fb_balkon_peryla_send(str_Rec:=fb_KL6301_0.str_Data_Rec, bData:=balkon_peryla,  Group_Address:=balkon_peryla_adr, bsend:=((fb_balkon_peryla_send.bData XOR fb_balkon_peryla_read.bData XOR balkon_peryla)OR fb_heartbeat2_timer.q));   (*       balkon_peryla_read.bData XOR balkon_peryla)) AND fb_heartbeat2_timer.q))      )));*)
IF NOT fb_balkon_peryla_read.bDataReceive OR  fb_heartbeat2_timer.q THEN fb_balkon_peryla_send.bSend:=FALSE; fb_balkon_peryla_send(str_Rec:=fb_KL6301_0.str_Data_Rec, bData:=balkon_peryla,  Group_Address:=balkon_peryla_adr);END_IF
fb_kino_l_send(str_Rec:=fb_KL6301_0.str_Data_Rec, bData:=kino_l,  Group_Address:=kino_l_adr, bsend:=((fb_kino_l_send.bData  <>  fb_kino_l_read.bData <> kino_l)OR fb_heartbeat2_timer.q));
IF NOT fb_kino_l_read.bDataReceive OR  fb_heartbeat2_timer.q THEN fb_kino_l_send.bSend:=FALSE; fb_kino_l_send(str_Rec:=fb_KL6301_0.str_Data_Rec,  Group_Address:=kino_l_adr);END_IF
fb_balkon_bra_send(str_Rec:=fb_KL6301_0.str_Data_Rec, bData:=balkon_bra,  Group_Address:=balkon_bra_adr, bsend:=((fb_balkon_bra_read.bData  XOR fb_balkon_bra_read.bData XOR balkon_bra)OR fb_heartbeat2_timer.q));   (*       balkon_bra_read.bData XOR balkon_bra)) AND fb_heartbeat2_timer.q))      )));*)
IF NOT fb_balkon_bra_read.bDataReceive OR  fb_heartbeat2_timer.q THEN fb_balkon_bra_send.bSend:=FALSE; fb_balkon_bra_send(str_Rec:=fb_KL6301_0.str_Data_Rec, bData:=balkon_bra,  Group_Address:=balkon_bra_adr);END_IF
fb_kabinet_balkon_l_send(str_Rec:=fb_KL6301_0.str_Data_Rec, bData:=kabinet_balkon_l,  Group_Address:=kabinet_balkon_l_adr, bsend:=(( fb_kabinet_balkon_l_send.bData XOR fb_kabinet_balkon_l_read.bData XOR kabinet_balkon_l)OR fb_heartbeat2_timer.q));   (*       kabinet_balkon_l_read.bData XOR kabinet_balkon_l)) AND fb_heartbeat2_timer.q))      )));*)
IF NOT fb_kabinet_balkon_l_read.bDataReceive OR  fb_heartbeat2_timer.q THEN fb_kabinet_balkon_l_send.bSend:=FALSE; fb_kabinet_balkon_l_send(str_Rec:=fb_KL6301_0.str_Data_Rec, bData:=kabinet_balkon_l,  Group_Address:=kabinet_balkon_l_adr);END_IF
fb_balkon_send(str_Rec:=fb_KL6301_0.str_Data_Rec, bData:=balkon,  Group_Address:=balkon_adr, bsend:=((fb_balkon_send.bData XOR fb_balkon_read.bData XOR balkon)OR fb_heartbeat2_timer.q));   (*       balkon_read.bData XOR balkon)) AND fb_heartbeat2_timer.q))      )));*)
IF NOT fb_balkon_read.bDataReceive OR  fb_heartbeat2_timer.q THEN fb_balkon_send.bSend:=FALSE; fb_balkon_send(str_Rec:=fb_KL6301_0.str_Data_Rec, bData:=balkon,  Group_Address:=balkon_adr);END_IF
fb_korydor1_send(str_Rec:=fb_KL6301_0.str_Data_Rec, bData:=korydor1,  Group_Address:=korydor1_adr, bsend:=((fb_korydor1_send.bData XOR fb_korydor1_read.bData XOR korydor1)OR fb_heartbeat2_timer.q));   (* *)
IF NOT fb_korydor1_read.bDataReceive OR  fb_heartbeat2_timer.q THEN fb_korydor1_send.bSend:=FALSE; fb_korydor1_send(str_Rec:=fb_KL6301_0.str_Data_Rec, bData:=korydor1,  Group_Address:=korydor1_adr);END_IF
fb_kino_bra_send(str_Rec:=fb_KL6301_0.str_Data_Rec, bData:=kino_bra,  Group_Address:=kino_bra_adr, bsend:=((fb_kino_bra_send.bData XOR fb_kino_bra_read.bData XOR kino_bra)OR fb_heartbeat2_timer.q));
IF NOT fb_kino_bra_read.bDataReceive OR  fb_heartbeat2_timer.q THEN fb_kino_bra_send.bSend:=FALSE; fb_kino_bra_send(str_Rec:=fb_KL6301_0.str_Data_Rec, bData:=kino_bra,  Group_Address:=kino_bra_adr);END_IF
fb_korydor2_send(str_Rec:=fb_KL6301_0.str_Data_Rec, bData:=korydor2,  Group_Address:=korydor2_adr, bsend:=((fb_korydor2_send.bData XOR fb_korydor2_read.bData XOR korydor2)OR fb_heartbeat2_timer.q));
IF NOT fb_korydor2_read.bDataReceive OR  fb_heartbeat2_timer.q THEN fb_korydor2_send.bSend:=FALSE; fb_korydor2_send(str_Rec:=fb_KL6301_0.str_Data_Rec, bData:=korydor2,  Group_Address:=korydor2_adr);END_IF
fb_studio_pidsvitka_send(str_Rec:=fb_KL6301_0.str_Data_Rec, bData:=studio_pidsvitka,  Group_Address:=studio_pidsvitka_adr, bsend:=((fb_studio_pidsvitka_send.bData XOR fb_studio_pidsvitka_read.bData XOR studio_pidsvitka)OR fb_heartbeat2_timer.q));
IF NOT fb_studio_pidsvitka_read.bDataReceive OR  fb_heartbeat2_timer.q THEN fb_studio_pidsvitka_send.bSend:=FALSE; fb_studio_pidsvitka_send(str_Rec:=fb_KL6301_0.str_Data_Rec, bData:=studio_pidsvitka,  Group_Address:=studio_pidsvitka_adr);END_IF
fb_skhody2_3_send(str_Rec:=fb_KL6301_0.str_Data_Rec, bData:=skhody2_3,  Group_Address:=skhody2_3_adr, bsend:=((fb_skhody2_3_send.bData XOR fb_skhody2_3_read.bData XOR skhody2_3)OR fb_heartbeat2_timer.q));
IF NOT fb_skhody2_3_read.bDataReceive OR  fb_heartbeat2_timer.q THEN fb_skhody2_3_send.bSend:=FALSE; fb_skhody2_3_send(str_Rec:=fb_KL6301_0.str_Data_Rec, bData:=skhody2_3,  Group_Address:=skhody2_3_adr);END_IF
fb_studio_l_send(str_Rec:=fb_KL6301_0.str_Data_Rec, bData:=studio_l,  Group_Address:=studio_l_adr, bsend:=((fb_studio_l_send.bData XOR fb_studio_l_read.bData XOR studio_l)OR fb_heartbeat2_timer.q));
IF NOT fb_studio_l_read.bDataReceive OR  fb_heartbeat2_timer.q THEN fb_studio_l_send.bSend:=FALSE; fb_studio_l_send(str_Rec:=fb_KL6301_0.str_Data_Rec, bData:=studio_l,  Group_Address:=studio_l_adr);END_IF
fb_kabinet_pidsvitka_kolo_send(str_Rec:=fb_KL6301_0.str_Data_Rec, bData:=kabinet_pidsvitka_kolo,  Group_Address:=kabinet_pidsvitka_kolo_adr, bsend:=((fb_kabinet_pidsvitka_kolo_send.bData XOR fb_kabinet_pidsvitka_kolo_read.bData XOR kabinet_pidsvitka_kolo)OR fb_heartbeat2_timer.q));
IF NOT fb_kabinet_pidsvitka_kolo_read.bDataReceive OR  fb_heartbeat2_timer.q THEN fb_kabinet_pidsvitka_kolo_send.bSend:=FALSE; fb_kabinet_pidsvitka_kolo_send(str_Rec:=fb_KL6301_0.str_Data_Rec, bData:=kabinet_pidsvitka_kolo,  Group_Address:=kabinet_pidsvitka_kolo_adr);END_IF
fb_kabinet_svitlo_send(str_Rec:=fb_KL6301_0.str_Data_Rec, bData:=kabinet_svitlo,  Group_Address:=kabinet_svitlo_adr, bsend:=((fb_kabinet_svitlo_send.bData XOR fb_kabinet_svitlo_read.bData XOR kabinet_svitlo)OR fb_heartbeat2_timer.q));
IF NOT fb_kabinet_svitlo_read.bDataReceive OR  fb_heartbeat2_timer.q THEN fb_kabinet_svitlo_send.bSend:=FALSE; fb_kabinet_svitlo_send(str_Rec:=fb_KL6301_0.str_Data_Rec, bData:=kabinet_svitlo,  Group_Address:=kabinet_svitlo_adr);END_IF
fb_stend_send(str_Rec:=fb_KL6301_0.str_Data_Rec, bData:=stend,  Group_Address:=stend_adr, bsend:=((fb_stend_send.bData XOR fb_stend_read.bData XOR stend)OR fb_heartbeat2_timer.q));
IF NOT fb_stend_read.bDataReceive OR  fb_heartbeat2_timer.q THEN fb_stend_send.bSend:=FALSE; fb_stend_send(str_Rec:=fb_KL6301_0.str_Data_Rec, bData:=stend,  Group_Address:=stend_adr);END_IF
fb_kabinet_kobra_send(str_Rec:=fb_KL6301_0.str_Data_Rec, bData:=kabinet_kobra,  Group_Address:=kabinet_kobra_adr, bsend:=((fb_kabinet_kobra_send.bData XOR fb_kabinet_kobra_read.bData XOR kabinet_kobra)OR fb_heartbeat2_timer.q));
IF NOT fb_kabinet_kobra_read.bDataReceive OR  fb_heartbeat2_timer.q THEN fb_kabinet_kobra_send.bSend:=FALSE; fb_kabinet_kobra_send(str_Rec:=fb_KL6301_0.str_Data_Rec, bData:=kabinet_kobra,  Group_Address:=kabinet_kobra_adr);END_IF
fb_skhody_peryla_send(str_Rec:=fb_KL6301_0.str_Data_Rec, bData:=skhody_peryla,  Group_Address:=skhody_peryla_adr, bsend:=((fb_skhody_peryla_send.bData XOR fb_skhody_peryla_read.bData XOR skhody_peryla)OR fb_heartbeat2_timer.q));
IF NOT fb_skhody_peryla_read.bDataReceive OR  fb_heartbeat2_timer.q THEN fb_skhody_peryla_send.bSend:=FALSE; fb_skhody_peryla_send(str_Rec:=fb_KL6301_0.str_Data_Rec, bData:=skhody_peryla,  Group_Address:=skhody_peryla_adr);END_IF
fb_tambur2_send(str_Rec:=fb_KL6301_0.str_Data_Rec, bData:=tambur2,  Group_Address:=tambur2_adr, bsend:=((fb_tambur2_send.bData XOR fb_tambur2_read.bData XOR tambur2)OR fb_heartbeat2_timer.q)) ;
IF NOT fb_tambur2_read.bDataReceive OR  fb_heartbeat2_timer.q THEN fb_tambur2_send.bSend:=FALSE; fb_tambur2_send(str_Rec:=fb_KL6301_0.str_Data_Rec, bData:=tambur2,  Group_Address:=tambur2_adr);END_IF

IF NOT  fb_balkon_peryla_read.bDataReceive THEN
	data2floor[100].0:=fb_balkon_peryla_read.bdata;
	balkon_peryla:=fb_balkon_peryla_read.bdata;
ELSE data2floor[100].0:=balkon_peryla; END_IF
IF NOT fb_kino_l_read.bDataReceive THEN
	data2floor[100].1:=fb_kino_l_read.bdata;
	kino_l:=fb_kino_l_read.bdata;
ELSE data2floor[100].1:=kino_l; END_IF
IF NOT fb_balkon_bra_read.bDataReceive THEN
	data2floor[100].2:= fb_balkon_bra_read.bdata;
	balkon_bra:= fb_balkon_bra_read.bdata;
ELSE data2floor[100].2:= balkon_bra;END_IF
IF NOT fb_kabinet_balkon_l_read.bDataReceive  THEN
	 data2floor[100].3:=fb_kabinet_balkon_l_read.bdata;
	kabinet_balkon_l:=fb_kabinet_balkon_l_read.bdata;
ELSE 	data2floor[100].3:=kabinet_balkon_l; END_IF
IF NOT fb_balkon_read.bDataReceive THEN
	data2floor[100].4:=fb_balkon_read.bdata;
	balkon:=fb_balkon_read.bdata;
ELSE 	data2floor[100].4:=balkon; END_IF
IF NOT fb_korydor1_read.bDataReceive THEN
	data2floor[100].5:=fb_korydor1_read.bdata;
	korydor1:=fb_korydor1_read.bdata;
ELSE 	data2floor[100].5:=korydor1;END_IF;
IF NOT fb_kino_bra_read.bDataReceive  THEN
	data2floor[100].6:=fb_kino_bra_read.bdata;
	kino_bra:=fb_kino_bra_read.bdata;
 ELSE 	data2floor[100].6:=kino_bra; END_IF;
IF NOT fb_korydor2_read.bDataReceive  THEN
	data2floor[100].7:=fb_korydor2_read.bdata;
	korydor2:=fb_korydor2_read.bdata;
ELSE 	data2floor[100].7:=korydor2; END_IF;
IF NOT fb_studio_pidsvitka_read.bDataReceive  THEN
	data2floor[101].0:=fb_studio_pidsvitka_read.bdata;
	studio_pidsvitka:=fb_studio_pidsvitka_read.bdata;
ELSE data2floor[101].0:=studio_pidsvitka; END_IF;
IF NOT fb_skhody2_3_read.bDataReceive  THEN
	data2floor[101].1:=fb_skhody2_3_read.bdata;
	skhody2_3:=fb_skhody2_3_read.bdata;
ELSE data2floor[101].1:=skhody2_3; END_IF;
IF NOT fb_studio_l_read.bDataReceive THEN
	data2floor[101].2:=fb_studio_l_read.bdata;
	studio_l:=fb_studio_l_read.bdata;
ELSE data2floor[101].2:=studio_l; END_IF;
IF NOT fb_kabinet_pidsvitka_kolo_read.bDataReceive THEN
	data2floor[101].3:=fb_kabinet_pidsvitka_kolo_read.bdata;
	kabinet_pidsvitka_kolo:=fb_kabinet_pidsvitka_kolo_read.bdata;
ELSE data2floor[101].3:=kabinet_pidsvitka_kolo; END_IF;
IF NOT fb_kabinet_svitlo_read.bDataReceive THEN
	data2floor[101].4:=fb_kabinet_svitlo_read.bdata;
	kabinet_svitlo:=fb_kabinet_svitlo_read.bdata;
ELSE data2floor[101].4:=kabinet_svitlo; END_IF;
IF NOT fb_kabinet_kobra_read.bDataReceive THEN
	data2floor[101].5:=fb_kabinet_kobra_read.bdata;
	kabinet_kobra:=fb_kabinet_kobra_read.bdata;
ELSE data2floor[101].5:=kabinet_kobra; END_IF;
IF NOT fb_tambur2_read.bDataReceive  THEN
	data2floor[101].6:=fb_tambur2_read.bdata;
	tambur2:=fb_tambur2_read.bdata;
ELSE data2floor[101].6:=tambur2; END_IF;
IF NOT fb_stend_read.bDataReceive  THEN
	data2floor[101].7:=fb_stend_read.bdata;
	stend:=fb_stend_read.bdata;
ELSE  data2floor[101].7:=stend; END_IF;
IF NOT fb_skhody_peryla_read.bDataReceive  THEN
	data2floor[102].0:=fb_skhody_peryla_read.bdata;
	skhody_peryla:=fb_skhody_peryla_read.bdata;
ELSE data2floor[102].0:=skhody_peryla; END_IF;
END_ACTION
ACTION floor3:
(*read*)
fb_spalnya_kontrazhur_read(strData_Rec:=fb_KL6301_0.str_Data_Rec, Group_Address:=spalnya_kontrazhur_adr);
fb_spalnya_balkon_read(strData_Rec:=fb_KL6301_0.str_Data_Rec,  Group_Address:=spalnya_balkon_adr);
fb_spalnya_kulbaba_read(strData_Rec:=fb_KL6301_0.str_Data_Rec, Group_Address:=spalnya_kulbaba_adr);
fb_spalnya_kontrazhur_b_read(strData_Rec:=fb_KL6301_0.str_Data_Rec, Group_Address:=spalnya_kontrazhur_b_adr);
fb_spalnya_kontrazhur_l_read(strData_Rec:=fb_KL6301_0.str_Data_Rec, Group_Address:=spalnya_kontrazhur_l_adr);
fb_su3_stina_read(strData_Rec:=fb_KL6301_0.str_Data_Rec, Group_Address:=su3_stina_adr);
fb_su3_pidsvitka_read(strData_Rec:=fb_KL6301_0.str_Data_Rec,  Group_Address:=su3_pidsvitka_adr);
fb_su3_bra_read(strData_Rec:=fb_KL6301_0.str_Data_Rec, Group_Address:=su3_bra_adr);
fb_su3_kontrazhur_read(strData_Rec:=fb_KL6301_0.str_Data_Rec, Group_Address:=su3_kontrazhur_adr);
fb_su3_kontrazhur_k_read(strData_Rec:=fb_KL6301_0.str_Data_Rec,  Group_Address:=su3_kontrazhur_k_adr);
fb_su3_lampa_read(strData_Rec:=fb_KL6301_0.str_Data_Rec, Group_Address:=su3_lampa_adr);
fb_dytjacha_read(strData_Rec:=fb_KL6301_0.str_Data_Rec, Group_Address:=dytjacha_adr);
fb_dytjacha_bra_read(strData_Rec:=fb_KL6301_0.str_Data_Rec, Group_Address:=dytjacha_bra_adr);
fb_garderob_read(strData_Rec:=fb_KL6301_0.str_Data_Rec, Group_Address:=garderob_adr);
fb_bar_read(strData_Rec:=fb_KL6301_0.str_Data_Rec, Group_Address:=bar_adr);
fb_korydor_skeli_read(strData_Rec:=fb_KL6301_0.str_Data_Rec, Group_Address:=korydor_skeli_adr);
fb_choven_read(strData_Rec:=fb_KL6301_0.str_Data_Rec, Group_Address:=choven_adr);
fb_korydor_lampa_read(strData_Rec:=fb_KL6301_0.str_Data_Rec, Group_Address:=korydor_lampa_adr);
fb_serverna_read(strData_Rec:=fb_KL6301_0.str_Data_Rec, Group_Address:=serverna_adr);
fb_korydor_svitlo_read(strData_Rec:=fb_KL6301_0.str_Data_Rec, Group_Address:=korydor_svitlo_adr);
fb_moove_sensors_read(strData_Rec:=fb_KL6301_0.str_Data_Rec, Group_Address:=moove_sensors_adr);

fb_spalnya_kontrazhur_send(str_Rec:=fb_KL6301_0.str_Data_Rec, bData:=spalnya_kontrazhur,  Group_Address:=spalnya_kontrazhur_adr, bsend:=((fb_spalnya_kontrazhur_send.bData XOR fb_spalnya_kontrazhur_read.bData XOR spalnya_kontrazhur)OR fb_heartbeat_timer.q));
IF NOT fb_spalnya_kontrazhur_read.bDataReceive OR  fb_heartbeat_timer.q THEN fb_spalnya_kontrazhur_send.bSend:=FALSE; fb_spalnya_kontrazhur_send(str_Rec:=fb_KL6301_0.str_Data_Rec, bData:=spalnya_kontrazhur,  Group_Address:=spalnya_kontrazhur_adr);END_IF
fb_spalnya_balkon_send(str_Rec:=fb_KL6301_0.str_Data_Rec, bData:=spalnya_balkon,  Group_Address:=spalnya_balkon_adr, bsend:=((fb_spalnya_balkon_send.bData XOR fb_spalnya_balkon_read.bData XOR spalnya_balkon)OR fb_heartbeat_timer.q));
IF NOT fb_spalnya_balkon_read.bDataReceive OR  fb_heartbeat_timer.q THEN fb_spalnya_balkon_send.bSend:=FALSE; fb_spalnya_balkon_send(str_Rec:=fb_KL6301_0.str_Data_Rec, bData:=spalnya_balkon,  Group_Address:=spalnya_balkon_adr);END_IF
fb_spalnya_kulbaba_send(str_Rec:=fb_KL6301_0.str_Data_Rec, bData:=spalnya_kulbaba,  Group_Address:=spalnya_kulbaba_adr, bsend:=((fb_spalnya_kulbaba_send.bData XOR fb_spalnya_kulbaba_read.bData XOR spalnya_kulbaba)OR fb_heartbeat_timer.q));
IF NOT fb_spalnya_kulbaba_read.bDataReceive OR  fb_heartbeat_timer.q THEN fb_spalnya_kulbaba_send.bSend:=FALSE; fb_spalnya_kulbaba_send(str_Rec:=fb_KL6301_0.str_Data_Rec, bData:=spalnya_kulbaba,  Group_Address:=spalnya_kulbaba_adr);END_IF
fb_spalnya_kontrazhur_b_send(str_Rec:=fb_KL6301_0.str_Data_Rec, bData:=spalnya_kontrazhur_b,  Group_Address:=spalnya_kontrazhur_b_adr, bsend:=((fb_spalnya_kontrazhur_b_send.bData XOR fb_spalnya_kontrazhur_b_read.bData XOR spalnya_kontrazhur_b)OR fb_heartbeat_timer.q));
IF NOT fb_spalnya_kontrazhur_b_read.bDataReceive OR  fb_heartbeat_timer.q THEN fb_spalnya_kontrazhur_b_send.bSend:=FALSE; fb_spalnya_kontrazhur_b_send(str_Rec:=fb_KL6301_0.str_Data_Rec, bData:=spalnya_kontrazhur_b,  Group_Address:=spalnya_kontrazhur_b_adr);END_IF
fb_spalnya_kontrazhur_l_send(str_Rec:=fb_KL6301_0.str_Data_Rec, bData:=spalnya_kontrazhur_l,  Group_Address:=spalnya_kontrazhur_l_adr, bsend:=((fb_spalnya_kontrazhur_l_send.bData XOR fb_spalnya_kontrazhur_l_read.bData XOR spalnya_kontrazhur_l)OR fb_heartbeat_timer.q));
IF NOT fb_spalnya_kontrazhur_l_read.bDataReceive OR  fb_heartbeat_timer.q THEN fb_spalnya_kontrazhur_l_send.bSend:=FALSE; fb_spalnya_kontrazhur_l_send(str_Rec:=fb_KL6301_0.str_Data_Rec, bData:=spalnya_kontrazhur_l,  Group_Address:=spalnya_kontrazhur_l_adr);END_IF
fb_su3_stina_send(str_Rec:=fb_KL6301_0.str_Data_Rec, bData:=su3_stina,  Group_Address:=su3_stina_adr, bsend:=((fb_su3_stina_send.bData XOR fb_su3_stina_read.bData XOR su3_stina)OR fb_heartbeat_timer.q));
IF NOT fb_su3_stina_read.bDataReceive OR  fb_heartbeat_timer.q THEN fb_su3_stina_send.bSend:=FALSE; fb_su3_stina_send(str_Rec:=fb_KL6301_0.str_Data_Rec, bData:=su3_stina,  Group_Address:=su3_stina_adr);END_IF
fb_su3_pidsvitka_send(str_Rec:=fb_KL6301_0.str_Data_Rec, bData:=su3_pidsvitka,  Group_Address:=su3_pidsvitka_adr, bsend:=((fb_su3_pidsvitka_send.bData XOR fb_su3_pidsvitka_read.bData XOR su3_pidsvitka)OR fb_heartbeat_timer.q));
IF NOT fb_su3_pidsvitka_read.bDataReceive OR  fb_heartbeat_timer.q THEN fb_su3_pidsvitka_send.bSend:=FALSE; fb_su3_pidsvitka_send(str_Rec:=fb_KL6301_0.str_Data_Rec, bData:=su3_pidsvitka,  Group_Address:=su3_pidsvitka_adr);END_IF
fb_su3_bra_send(str_Rec:=fb_KL6301_0.str_Data_Rec, bData:=su3_bra,  Group_Address:=su3_bra_adr, bsend:=((fb_su3_bra_send.bData XOR fb_su3_bra_read.bData XOR su3_bra)OR fb_heartbeat_timer.q));
IF NOT fb_su3_bra_read.bDataReceive OR  fb_heartbeat_timer.q THEN fb_su3_bra_send.bSend:=FALSE; fb_su3_bra_send(str_Rec:=fb_KL6301_0.str_Data_Rec, bData:=su3_bra,  Group_Address:=su3_bra_adr);END_IF
fb_su3_kontrazhur_send(str_Rec:=fb_KL6301_0.str_Data_Rec, bData:=su3_kontrazhur,  Group_Address:=su3_kontrazhur_adr, bsend:=((fb_su3_kontrazhur_send.bData XOR fb_su3_kontrazhur_read.bData XOR su3_kontrazhur)OR fb_heartbeat_timer.q));
IF NOT fb_su3_kontrazhur_read.bDataReceive OR  fb_heartbeat_timer.q THEN fb_su3_kontrazhur_send.bSend:=FALSE; fb_su3_kontrazhur_send(str_Rec:=fb_KL6301_0.str_Data_Rec, bData:=su3_kontrazhur,  Group_Address:=su3_kontrazhur_adr);END_IF
fb_su3_kontrazhur_k_send(str_Rec:=fb_KL6301_0.str_Data_Rec, bData:=su3_kontrazhur_k,  Group_Address:=su3_kontrazhur_k_adr, bsend:=((fb_su3_kontrazhur_k_send.bData XOR fb_su3_kontrazhur_k_read.bData XOR su3_kontrazhur_k)OR fb_heartbeat_timer.q));
IF NOT fb_su3_kontrazhur_k_read.bDataReceive OR  fb_heartbeat_timer.q THEN fb_su3_kontrazhur_k_send.bSend:=FALSE; fb_su3_kontrazhur_k_send(str_Rec:=fb_KL6301_0.str_Data_Rec, bData:=su3_kontrazhur_k,  Group_Address:=su3_kontrazhur_k_adr);END_IF
fb_su3_lampa_send(str_Rec:=fb_KL6301_0.str_Data_Rec, bData:=su3_lampa,  Group_Address:=su3_lampa_adr, bsend:=((fb_su3_lampa_send.bData XOR fb_su3_lampa_read.bData XOR su3_lampa)OR fb_heartbeat_timer.q));
IF NOT fb_su3_lampa_read.bDataReceive OR  fb_heartbeat_timer.q THEN fb_su3_lampa_send.bSend:=FALSE; fb_su3_lampa_send(str_Rec:=fb_KL6301_0.str_Data_Rec, bData:=su3_lampa,  Group_Address:=su3_lampa_adr);END_IF
fb_dytjacha_send(str_Rec:=fb_KL6301_0.str_Data_Rec, bData:=dytjacha,  Group_Address:=dytjacha_adr, bsend:=((fb_dytjacha_send.bData XOR fb_dytjacha_read.bData XOR dytjacha)OR fb_heartbeat_timer.q));
IF NOT fb_dytjacha_read.bDataReceive OR  fb_heartbeat_timer.q THEN fb_dytjacha_send.bSend:=FALSE; fb_dytjacha_send(str_Rec:=fb_KL6301_0.str_Data_Rec, bData:=dytjacha,  Group_Address:=dytjacha_adr);END_IF
fb_dytjacha_bra_send(str_Rec:=fb_KL6301_0.str_Data_Rec, bData:=dytjacha_bra,  Group_Address:=dytjacha_bra_adr, bsend:=((fb_dytjacha_bra_send.bData XOR fb_dytjacha_bra_read.bData XOR dytjacha_bra)OR fb_heartbeat_timer.q));
IF NOT fb_dytjacha_bra_read.bDataReceive OR  fb_heartbeat_timer.q THEN fb_dytjacha_bra_send.bSend:=FALSE; fb_dytjacha_bra_send(str_Rec:=fb_KL6301_0.str_Data_Rec, bData:=dytjacha_bra,  Group_Address:=dytjacha_bra_adr);END_IF
fb_garderob_send(str_Rec:=fb_KL6301_0.str_Data_Rec, bData:=garderob,  Group_Address:=garderob_adr, bsend:=((fb_garderob_read.bData XOR garderob XOR fb_garderob_send.bData )OR fb_heartbeat_timer.q));
IF NOT fb_garderob_read.bDataReceive OR  fb_heartbeat_timer.q THEN fb_garderob_send.bSend:=FALSE; fb_garderob_send(str_Rec:=fb_KL6301_0.str_Data_Rec, bData:=garderob,  Group_Address:=garderob_adr);END_IF
fb_bar_send(str_Rec:=fb_KL6301_0.str_Data_Rec, bData:=bar,  Group_Address:=bar_adr, bsend:=((fb_bar_send.bData XOR fb_bar_read.bData XOR bar)OR fb_heartbeat_timer.q));
IF NOT fb_bar_read.bDataReceive OR  fb_heartbeat_timer.q THEN fb_bar_send.bSend:=FALSE; fb_bar_send(str_Rec:=fb_KL6301_0.str_Data_Rec, bData:=bar,  Group_Address:=bar_adr);END_IF
fb_korydor_skeli_send(str_Rec:=fb_KL6301_0.str_Data_Rec, bData:=korydor_skeli,  Group_Address:=korydor_skeli_adr, bsend:=((fb_korydor_skeli_read.bData XOR korydor_skeli XOR fb_korydor_skeli_send.bData )OR fb_heartbeat_timer.q));
IF  NOT fb_korydor_skeli_read.bDataReceive OR  fb_heartbeat_timer.q THEN  fb_korydor_skeli_send.bSend:=FALSE; fb_korydor_skeli_send(str_Rec:=fb_KL6301_0.str_Data_Rec, bData:=korydor_skeli,  Group_Address:=korydor_skeli_adr);END_IF
fb_choven_send(str_Rec:=fb_KL6301_0.str_Data_Rec, bData:=choven,  Group_Address:=choven_adr, bsend:=((fb_choven_read.bData XOR choven XOR fb_choven_send.bData )OR fb_heartbeat_timer.q));
IF NOT fb_choven_read.bDataReceive OR  fb_heartbeat_timer.q THEN fb_choven_send.bSend:=FALSE; fb_choven_send(str_Rec:=fb_KL6301_0.str_Data_Rec, bData:=choven,  Group_Address:=choven_adr);END_IF
fb_korydor_svitlo_send(str_Rec:=fb_KL6301_0.str_Data_Rec, bData:=korydor_svitlo,  Group_Address:=korydor_svitlo_adr, bsend:=((fb_korydor_svitlo_send.bData XOR fb_korydor_svitlo_read.bData XOR korydor_svitlo)OR fb_heartbeat_timer.q));
IF NOT fb_korydor_svitlo_read.bDataReceive OR  fb_heartbeat_timer.q THEN fb_korydor_svitlo_send.bSend:=FALSE; fb_korydor_svitlo_send(str_Rec:=fb_KL6301_0.str_Data_Rec, bData:=korydor_svitlo,  Group_Address:=korydor_svitlo_adr);END_IF
fb_korydor_lampa_send(str_Rec:=fb_KL6301_0.str_Data_Rec, bData:=korydor_lampa,  Group_Address:=korydor_lampa_adr, bsend:=((fb_korydor_lampa_read.bData XOR korydor_lampa XOR fb_korydor_lampa_send.bData )OR fb_heartbeat_timer.q));
IF NOT fb_korydor_lampa_read.bDataReceive OR  fb_heartbeat_timer.q THEN fb_korydor_lampa_send.bSend:=FALSE; fb_korydor_lampa_send(str_Rec:=fb_KL6301_0.str_Data_Rec, bData:=korydor_lampa,  Group_Address:=korydor_lampa_adr);END_IF
fb_serverna_send(str_Rec:=fb_KL6301_0.str_Data_Rec, bData:=serverna,  Group_Address:=serverna_adr, bsend:=((fb_serverna_send.bData XOR fb_serverna_read.bData XOR serverna)OR fb_heartbeat_timer.q));
IF NOT fb_serverna_read.bDataReceive OR  fb_heartbeat_timer.q THEN fb_serverna_send.bSend:=FALSE; fb_serverna_send(str_Rec:=fb_KL6301_0.str_Data_Rec, bData:=serverna,  Group_Address:=serverna_adr);END_IF
END_ACTION
ACTION PanelBus:
CASE fb_kl6301_0.GroupReceive.SUB_MAIN OF
	1:(*vitalnya*)
	IF fb_kl6301_0.GroupReceive.number <10 AND fb_kl6301_0.GroupReceive.number <>0 THEN vitalnya_hvac.heat_mode:=fb_kl6301_0.GroupReceive.number;END_IF
		CASE fb_kl6301_0.GroupReceive.number OF
			0:		fb_temp_read(Group_Address:=vitalnya_T_EIB_addr, strData_Rec:=fb_KL6301_0.str_Data_Rec, rData=>Vitalnya_HVAC.cur_t); (*temperature*)
			1:		fb_setpoint_read(Group_address:=vitalnya_cooling_EIB_addr, strData_Rec:=fb_KL6301_0.str_Data_Rec, byData=>setpoint_vitalnya_dpt4 ); (*cooling*)
					CASE REAL_TO_INT(setpoint_vitalnya_dpt4*100/255.0) OF
						0..30:		vitalnya_hvac.heat_speed:=1;
									vitalnya_hvac.t_ust_cool:= REAL_TO_INT(setpoint_vitalnya_dpt4*100/255.0); (*low speed*)
						31..59:		vitalnya_hvac.heat_speed:=2;
									vitalnya_hvac.t_ust_cool:= REAL_TO_INT(setpoint_vitalnya_dpt4*100/255.0-30); (*med speed*)
						60..100:	vitalnya_hvac.heat_speed:=3;
									vitalnya_hvac.t_ust_cool:= REAL_TO_INT(setpoint_vitalnya_dpt4*100/255.0-60); (*high speed*)
					END_CASE
					vitalnya_hvac.cur_t_ust:=vitalnya_hvac.t_ust_cool;
					(*
					надсилання в мережу прийнятого значення завдання
					fb_actual_setpoint_send(group_address:=vitalnya_actual_setpoint_addr, str_Rec:=fb_kl6301_0.str_Data_Rec, rData:=vitalnya_hvac.cur_t_ust);
					*)
			2:		fb_setpoint_read(Group_address:=vitalnya_heating_EIB_addr, strData_Rec:=fb_KL6301_0.str_Data_Rec, byData=>setpoint_vitalnya_dpt4 );  (*heating*)
					CASE REAL_TO_INT(setpoint_vitalnya_dpt4*100/255.0) OF
						0..30:		vitalnya_hvac.heat_speed:=1;
									vitalnya_hvac.t_ust_heat:= REAL_TO_INT(setpoint_vitalnya_dpt4*100/255.0); (*low speed*)
						31..59:		vitalnya_hvac.heat_speed:=2;
									vitalnya_hvac.t_ust_heat:= REAL_TO_INT(setpoint_vitalnya_dpt4*100/255.0-30); (*med speed*)
						60..100:	vitalnya_hvac.heat_speed:=3;
									vitalnya_hvac.t_ust_heat:= REAL_TO_INT(setpoint_vitalnya_dpt4*100/255.0-60); (*high speed*)
					END_CASE
					vitalnya_hvac.cur_t_ust:=vitalnya_hvac.t_ust_heat;
					(*
					fb_actual_setpoint_send(group_address:=vitalnya_actual_setpoint_addr, str_Rec:=fb_kl6301_0.str_Data_Rec, rData:=vitalnya_hvac.cur_t_ust);
					*)
			3:		fb_setpoint_read(Group_address:=vitalnya_fan_EIB_addr, strData_Rec:=fb_KL6301_0.str_Data_Rec, byData=>fanspeed_dpt4);
					VITALNYA_HVAC.heat_speed:=REAL_TO_USINT(fanspeed_dpt4*100/255.0);
			4:		VITALNYA_HVAC.heat_mode:=0;
			5:		fb_actual_setpoint_read(Group_Address:=vitalnya_actual_setpoint_addr, strData_Rec:=fb_KL6301_0.str_Data_Rec );
					vitalnya_hvac.cur_t_ust:=fb_actual_setpoint_read.rData;
		END_CASE;
	2: ;(*kino*)
	IF fb_kl6301_0.GroupReceive.number <10 AND fb_kl6301_0.GroupReceive.number <>0 THEN kino_hvac.heat_mode:=fb_kl6301_0.GroupReceive.number;END_IF
		CASE fb_kl6301_0.GroupReceive.number OF
			0:		fb_temp_read(Group_Address:=kino_T_EIB_addr, strData_Rec:=fb_KL6301_0.str_Data_Rec, rData=>kino_HVAC.cur_t); (*temperature*)
			1:		fb_setpoint_read(Group_address:=kino_cooling_EIB_addr, strData_Rec:=fb_KL6301_0.str_Data_Rec, byData=>setpoint_kino_dpt4 ); (*cooling*)
					CASE REAL_TO_INT(setpoint_kino_dpt4*100/255.0) OF
						0..30:		kino_hvac.heat_speed:=1;
									kino_hvac.t_ust_cool:= REAL_TO_INT(setpoint_kino_dpt4*100/255.0); (*low speed*)
						31..59:		kino_hvac.heat_speed:=2;
									kino_hvac.t_ust_cool:= REAL_TO_INT(setpoint_kino_dpt4*100/255.0-30); (*med speed*)
						60..100:	kino_hvac.heat_speed:=3;
									kino_hvac.t_ust_cool:= REAL_TO_INT(setpoint_kino_dpt4*100/255.0-60); (*high speed*)
					END_CASE
					kino_hvac.cur_t_ust:=kino_hvac.t_ust_cool;
					(*fb_actual_setpoint_send(group_address:=kino_actual_setpoint_addr, str_Rec:=fb_kl6301_0.str_Data_Rec, rData:=kino_hvac.cur_t_ust);*)
					kino_HVAc.manual_mode:=0;

			2:		fb_setpoint_read(Group_address:=kino_heating_EIB_addr, strData_Rec:=fb_KL6301_0.str_Data_Rec, byData=>setpoint_kino_dpt4 );  (*heating*)
					CASE REAL_TO_INT(setpoint_kino_dpt4*100/255.0) OF
						0..30:		kino_hvac.heat_speed:=1;
									kino_hvac.t_ust_heat:= REAL_TO_INT(setpoint_kino_dpt4*100/255.0); (*low speed*)
						31..59:		kino_hvac.heat_speed:=2;
									kino_hvac.t_ust_heat:= REAL_TO_INT(setpoint_kino_dpt4*100/255.0-30); (*med speed*)
						60..100:	kino_hvac.heat_speed:=3;
									kino_hvac.t_ust_heat:= REAL_TO_INT(setpoint_kino_dpt4*100/255.0-60); (*high speed*)
					END_CASE
					kino_hvac.cur_t_ust:=kino_hvac.t_ust_heat;
					(*fb_actual_setpoint_send(group_address:=kino_actual_setpoint_addr, str_Rec:=fb_kl6301_0.str_Data_Rec, rData:=kino_hvac.cur_t_ust);*)
					kino_HVAc.manual_mode:=0;
			3:		fb_setpoint_read(Group_address:=kino_fan_EIB_addr, strData_Rec:=fb_KL6301_0.str_Data_Rec, byData=>fanspeed_dpt4);
					kino_HVAC.heat_speed:=REAL_TO_USINT(fanspeed_dpt4*100/255.0);
					kino_HVAc.manual_mode:=0;
			4:		KINO_HVAC .heat_mode:=0; kino_HVAc.manual_mode:=1;
			5:		fb_actual_setpoint_read(Group_Address:=kino_actual_setpoint_addr, strData_Rec:=fb_KL6301_0.str_Data_Rec );
					kino_hvac.cur_t_ust:=fb_actual_setpoint_read.rData;
					kino_HVAc.manual_mode:=0;

		END_CASE;

	3: ;(*studio*)
	IF fb_kl6301_0.GroupReceive.number <10 AND fb_kl6301_0.GroupReceive.number <>0 THEN studio_hvac.heat_mode:=fb_kl6301_0.GroupReceive.number;END_IF
		CASE fb_kl6301_0.GroupReceive.number OF
			0:		fb_temp_read(Group_Address:=studio_T_EIB_addr, strData_Rec:=fb_KL6301_0.str_Data_Rec, rData=>studio_HVAC.cur_t); (*temperature*)
			1:		fb_setpoint_read(Group_address:=studio_cooling_EIB_addr, strData_Rec:=fb_KL6301_0.str_Data_Rec, byData=>setpoint_studio_dpt4 ); (*cooling*)
					CASE REAL_TO_INT(setpoint_studio_dpt4*100/255.0) OF
						0..30:		studio_hvac.heat_speed:=1;
									studio_hvac.t_ust_cool:= REAL_TO_INT(setpoint_studio_dpt4*100/255.0); (*low speed*)
						31..59:		studio_hvac.heat_speed:=2;
									studio_hvac.t_ust_cool:= REAL_TO_INT(setpoint_studio_dpt4*100/255.0-30); (*med speed*)
						60..100:	studio_hvac.heat_speed:=3;
									studio_hvac.t_ust_cool:= REAL_TO_INT(setpoint_studio_dpt4*100/255.0-60); (*high speed*)
					END_CASE
					studio_hvac.cur_t_ust:=studio_hvac.t_ust_cool;
					(*fb_actual_setpoint_send(group_address:=studio_actual_setpoint_addr, str_Rec:=fb_kl6301_0.str_Data_Rec, rData:=studio_hvac.cur_t_ust);*)

			2:		fb_setpoint_read(Group_address:=studio_heating_EIB_addr, strData_Rec:=fb_KL6301_0.str_Data_Rec, byData=>setpoint_studio_dpt4 );  (*heating*)
					CASE REAL_TO_INT(setpoint_studio_dpt4*100/255.0) OF
						0..30:		studio_hvac.heat_speed:=1;
									studio_hvac.t_ust_heat:= REAL_TO_INT(setpoint_studio_dpt4*100/255.0); (*low speed*)
						31..59:		studio_hvac.heat_speed:=2;
									studio_hvac.t_ust_heat:= REAL_TO_INT(setpoint_studio_dpt4*100/255.0-30); (*med speed*)
						60..100:	studio_hvac.heat_speed:=3;
									studio_hvac.t_ust_heat:= REAL_TO_INT(setpoint_studio_dpt4*100/255.0-60); (*high speed*)
					END_CASE
					studio_hvac.cur_t_ust:=studio_hvac.t_ust_heat;
					(*fb_actual_setpoint_send(group_address:=studio_actual_setpoint_addr, str_Rec:=fb_kl6301_0.str_Data_Rec, rData:=studio_hvac.cur_t_ust);*)

			3:		fb_setpoint_read(Group_address:=studio_fan_EIB_addr, strData_Rec:=fb_KL6301_0.str_Data_Rec, byData=>fanspeed_dpt4);
					studio_HVAC.heat_speed:=REAL_TO_USINT(fanspeed_dpt4*100/255.0);
			4:		STUDIO_HVAC.heat_mode:=0;
			5:		fb_actual_setpoint_read(Group_Address:=studio_actual_setpoint_addr, strData_Rec:=fb_KL6301_0.str_Data_Rec );
					studio_hvac.cur_t_ust:=fb_actual_setpoint_read.rData;

		END_CASE;

	4: ;(*kabinet*)
		IF fb_kl6301_0.GroupReceive.number <10 AND fb_kl6301_0.GroupReceive.number <>0 THEN kabinet_hvac.heat_mode:=fb_kl6301_0.GroupReceive.number;END_IF
		CASE fb_kl6301_0.GroupReceive.number OF
			0:		fb_temp_read(Group_Address:=kabinet_T_EIB_addr, strData_Rec:=fb_KL6301_0.str_Data_Rec, rData=>kabinet_HVAC.cur_t); (*temperature*)
			1:		fb_setpoint_read(Group_address:=kabinet_cooling_EIB_addr, strData_Rec:=fb_KL6301_0.str_Data_Rec, byData=>setpoint_kabinet_dpt4 ); (*cooling*)
					CASE REAL_TO_INT(setpoint_kabinet_dpt4*100/255.0) OF
						0..30:		kabinet_hvac.heat_speed:=1;
									kabinet_hvac.t_ust_cool:= REAL_TO_INT(setpoint_kabinet_dpt4*100/255.0); (*low speed*)
						31..59:		kabinet_hvac.heat_speed:=2;
									kabinet_hvac.t_ust_cool:= REAL_TO_INT(setpoint_kabinet_dpt4*100/255.0-30); (*med speed*)
						60..100:	kabinet_hvac.heat_speed:=3;
									kabinet_hvac.t_ust_cool:= REAL_TO_INT(setpoint_kabinet_dpt4*100/255.0-60); (*high speed*)
					END_CASE
					kabinet_hvac.cur_t_ust:=kabinet_hvac.t_ust_cool;
					(*fb_actual_setpoint_send(group_address:=kabinet_actual_setpoint_addr, str_Rec:=fb_kl6301_0.str_Data_Rec, rData:=kabinet_hvac.cur_t_ust);*)

			2:		fb_setpoint_read(Group_address:=kabinet_heating_EIB_addr, strData_Rec:=fb_KL6301_0.str_Data_Rec, byData=>setpoint_kabinet_dpt4 );  (*heating*)
					CASE REAL_TO_INT(setpoint_kabinet_dpt4*100/255.0) OF
						0..30:		kabinet_hvac.heat_speed:=1;
									kabinet_hvac.t_ust_heat:= REAL_TO_INT(setpoint_kabinet_dpt4*100/255.0); (*low speed*)
						31..59:		kabinet_hvac.heat_speed:=2;
									kabinet_hvac.t_ust_heat:= REAL_TO_INT(setpoint_kabinet_dpt4*100/255.0-30); (*med speed*)
						60..100:	kabinet_hvac.heat_speed:=3;
									kabinet_hvac.t_ust_heat:= REAL_TO_INT(setpoint_kabinet_dpt4*100/255.0-60); (*high speed*)
					END_CASE
					kabinet_hvac.cur_t_ust:=kabinet_hvac.t_ust_heat;
					(*fb_actual_setpoint_send(group_address:=kabinet_actual_setpoint_addr, str_Rec:=fb_kl6301_0.str_Data_Rec, rData:=kabinet_hvac.cur_t_ust);*)


			3:		fb_setpoint_read(Group_address:=kabinet_fan_EIB_addr, strData_Rec:=fb_KL6301_0.str_Data_Rec, byData=>fanspeed_dpt4);
					kabinet_HVAC.heat_speed:=REAL_TO_USINT(fanspeed_dpt4*100/255.0);
			4:		KABINET_HVAC.heat_mode:=0;
			5:		fb_actual_setpoint_read(Group_Address:=kabinet_actual_setpoint_addr, strData_Rec:=fb_KL6301_0.str_Data_Rec );
					kabinet_hvac.cur_t_ust:=fb_actual_setpoint_read.rData;

		END_CASE;

	5: ;(*dytjacha*)
		IF fb_kl6301_0.GroupReceive.number <10 AND fb_kl6301_0.GroupReceive.number <>0 THEN dytjacha_hvac.heat_mode:=fb_kl6301_0.GroupReceive.number;END_IF
		CASE fb_kl6301_0.GroupReceive.number OF
			0:		fb_temp_read(Group_Address:=dytjacha_T_EIB_addr, strData_Rec:=fb_KL6301_0.str_Data_Rec, rData=>dytjacha_HVAC.cur_t); (*temperature*)
			1:		fb_setpoint_read(Group_address:=dytjacha_cooling_EIB_addr, strData_Rec:=fb_KL6301_0.str_Data_Rec, byData=>setpoint_dytjacha_dpt4 ); (*cooling*)
					CASE REAL_TO_INT(setpoint_dytjacha_dpt4*100/255.0) OF
						0..30:		dytjacha_hvac.heat_speed:=1;
									dytjacha_hvac.t_ust_cool:= REAL_TO_INT(setpoint_dytjacha_dpt4*100/255.0); (*low speed*)
						31..59:		dytjacha_hvac.heat_speed:=2;
									dytjacha_hvac.t_ust_cool:= REAL_TO_INT(setpoint_dytjacha_dpt4*100/255.0-30); (*med speed*)
						60..100:	dytjacha_hvac.heat_speed:=3;
									dytjacha_hvac.t_ust_cool:= REAL_TO_INT(setpoint_dytjacha_dpt4*100/255.0-60); (*high speed*)
					END_CASE
					dytjacha_hvac.cur_t_ust:=dytjacha_hvac.t_ust_cool;
					(*fb_actual_setpoint_send(group_address:=dytjacha_actual_setpoint_addr, str_Rec:=fb_kl6301_0.str_Data_Rec, rData:=dytjacha_hvac.cur_t_ust);*)

			2:		fb_setpoint_read(Group_address:=dytjacha_heating_EIB_addr, strData_Rec:=fb_KL6301_0.str_Data_Rec, byData=>setpoint_dytjacha_dpt4 );  (*heating*)
					CASE REAL_TO_INT(setpoint_dytjacha_dpt4*100/255.0) OF
						0..30:		dytjacha_hvac.heat_speed:=1;
									dytjacha_hvac.t_ust_heat:= REAL_TO_INT(setpoint_dytjacha_dpt4*100/255.0); (*low speed*)
						31..59:		dytjacha_hvac.heat_speed:=2;
									dytjacha_hvac.t_ust_heat:= REAL_TO_INT(setpoint_dytjacha_dpt4*100/255.0-30); (*med speed*)
						60..100:	dytjacha_hvac.heat_speed:=3;
									dytjacha_hvac.t_ust_heat:= REAL_TO_INT(setpoint_dytjacha_dpt4*100/255.0-60); (*high speed*)
					END_CASE
					dytjacha_hvac.cur_t_ust:=dytjacha_hvac.t_ust_heat;
					(*fb_actual_setpoint_send(group_address:=dytjacha_actual_setpoint_addr, str_Rec:=fb_kl6301_0.str_Data_Rec, rData:=dytjacha_hvac.cur_t_ust);*)


			3:		fb_setpoint_read(Group_address:=dytjacha_fan_EIB_addr, strData_Rec:=fb_KL6301_0.str_Data_Rec, byData=>fanspeed_dpt4);
					dytjacha_HVAC.heat_speed:=REAL_TO_USINT(fanspeed_dpt4*100/255.0);
			4:		DYTJACHA_HVAC.heat_mode:=0;
			5:		fb_actual_setpoint_read(Group_Address:=dytjacha_actual_setpoint_addr, strData_Rec:=fb_KL6301_0.str_Data_Rec );
					dytjacha_hvac.cur_t_ust:=fb_actual_setpoint_read.rData;

		END_CASE;

	6: ;(*spalnya*)
		IF fb_kl6301_0.GroupReceive.number <10 AND fb_kl6301_0.GroupReceive.number <>0 THEN spalnya_hvac.heat_mode:=fb_kl6301_0.GroupReceive.number;END_IF
		CASE fb_kl6301_0.GroupReceive.number OF
			0:		fb_temp_read(Group_Address:=spalnya_T_EIB_addr, strData_Rec:=fb_KL6301_0.str_Data_Rec, rData=>spalnya_HVAC.cur_t); (*temperature*)
			1:		fb_setpoint_read(Group_address:=spalnya_cooling_EIB_addr, strData_Rec:=fb_KL6301_0.str_Data_Rec, byData=>setpoint_spalnya_dpt4 ); (*cooling*)
					CASE REAL_TO_INT(setpoint_spalnya_dpt4*100/255.0) OF
						0..30:		spalnya_hvac.heat_speed:=1;
									spalnya_hvac.t_ust_cool:= REAL_TO_INT(setpoint_spalnya_dpt4*100/255.0); (*low speed*)
						31..59:		spalnya_hvac.heat_speed:=2;
									spalnya_hvac.t_ust_cool:= REAL_TO_INT(setpoint_spalnya_dpt4*100/255.0-30); (*med speed*)
						60..100:	spalnya_hvac.heat_speed:=3;
									spalnya_hvac.t_ust_cool:= REAL_TO_INT(setpoint_spalnya_dpt4*100/255.0-60); (*high speed*)
					END_CASE
					spalnya_hvac.cur_t_ust:=spalnya_hvac.t_ust_cool;
					(*fb_actual_setpoint_send(group_address:=spalnya_actual_setpoint_addr, str_Rec:=fb_kl6301_0.str_Data_Rec, rData:=spalnya_hvac.cur_t_ust);*)

			2:		fb_setpoint_read(Group_address:=spalnya_heating_EIB_addr, strData_Rec:=fb_KL6301_0.str_Data_Rec, byData=>setpoint_spalnya_dpt4 );  (*heating*)
					CASE REAL_TO_INT(setpoint_spalnya_dpt4*100/255.0) OF
						0..30:		spalnya_hvac.heat_speed:=1;
									spalnya_hvac.t_ust_heat:= REAL_TO_INT(setpoint_spalnya_dpt4*100/255.0); (*low speed*)
						31..59:		spalnya_hvac.heat_speed:=2;
									spalnya_hvac.t_ust_heat:= REAL_TO_INT(setpoint_spalnya_dpt4*100/255.0-30); (*med speed*)
						60..100:	spalnya_hvac.heat_speed:=3;
									spalnya_hvac.t_ust_heat:= REAL_TO_INT(setpoint_spalnya_dpt4*100/255.0-60); (*high speed*)
					END_CASE
					spalnya_hvac.cur_t_ust:=spalnya_hvac.t_ust_heat;
					(*fb_actual_setpoint_send(group_address:=spalnya_actual_setpoint_addr, str_Rec:=fb_kl6301_0.str_Data_Rec, rData:=spalnya_hvac.cur_t_ust);*)


			3:		fb_setpoint_read(Group_address:=spalnya_fan_EIB_addr, strData_Rec:=fb_KL6301_0.str_Data_Rec, byData=>fanspeed_dpt4);
					spalnya_HVAC.heat_speed:=REAL_TO_USINT(fanspeed_dpt4*100/255.0);
			4:		SPALNYA_HVAC.heat_mode:=0;
			5:		fb_actual_setpoint_read(Group_Address:=spalnya_actual_setpoint_addr, strData_Rec:=fb_KL6301_0.str_Data_Rec );
					spalnya_hvac.cur_t_ust:=fb_actual_setpoint_read.rData;

		END_CASE;
END_CASE



(*hdl gate can transmit 2byte values, but they can not be assigned to DLP panel AC unit setpoint value directly,
so for every setpoint value in range [20,30] a 1 bit eib telegram with corresponding  adress +100 ( [120,130] ) should be generated and transmitted to HDL logic module and then
logic module assigns it to apropriate value DLP panel AC unit. 
amen*)
fb_setpoint_switch_send.iMode:=2;
fb_setpoint_switch_send.bStart:=TRUE;
IF vitalnya_hvac.cur_t_ust_prev <> vitalnya_hvac.cur_t_ust THEN
	fb_setpoint_switch_send.Group_Address.NUMBER:=REAL_TO_BYTE(vitalnya_hvac.cur_t_ust)+100;
	fb_setpoint_switch_send.Group_Address.MAIN:=1;
	fb_setpoint_switch_send.Group_Address.SUB_MAIN:=1;
	fb_setpoint_switch_send(str_Rec:=fb_KL6301_0.str_Data_Rec, bData:=FALSE);
	fb_setpoint_switch_send(str_Rec:=fb_KL6301_0.str_Data_Rec, bData:=TRUE);
END_IF
IF kino_hvac.cur_t_ust_prev <> kino_hvac.cur_t_ust THEN
	fb_setpoint_switch_send.Group_Address.NUMBER:=REAL_TO_BYTE(kino_hvac.cur_t_ust)+100;
	fb_setpoint_switch_send.Group_Address.MAIN:=1;
	fb_setpoint_switch_send.Group_Address.SUB_MAIN:=2;
	fb_setpoint_switch_send(str_Rec:=fb_KL6301_0.str_Data_Rec, bData:=1);
	fb_setpoint_switch_send(str_Rec:=fb_KL6301_0.str_Data_Rec, bData:=0);
END_IF
IF studio_hvac.cur_t_ust_prev <> studio_hvac.cur_t_ust THEN
	fb_setpoint_switch_send.Group_Address.NUMBER:=REAL_TO_BYTE(studio_hvac.cur_t_ust)+100;
	fb_setpoint_switch_send.Group_Address.MAIN:=1;
	fb_setpoint_switch_send.Group_Address.SUB_MAIN:=3;
	fb_setpoint_switch_send(str_Rec:=fb_KL6301_0.str_Data_Rec, bData:=1);
	fb_setpoint_switch_send(str_Rec:=fb_KL6301_0.str_Data_Rec, bData:=0);
END_IF
IF kabinet_hvac.cur_t_ust_prev <> kabinet_hvac.cur_t_ust THEN
	fb_setpoint_switch_send.Group_Address.NUMBER:=REAL_TO_BYTE(kabinet_hvac.cur_t_ust)+100;
	fb_setpoint_switch_send.Group_Address.MAIN:=1;
	fb_setpoint_switch_send.Group_Address.SUB_MAIN:=4;
	fb_setpoint_switch_send(str_Rec:=fb_KL6301_0.str_Data_Rec, bData:=1);
	fb_setpoint_switch_send(str_Rec:=fb_KL6301_0.str_Data_Rec, bData:=0);
END_IF
IF dytjacha_hvac.cur_t_ust_prev <> dytjacha_hvac.cur_t_ust THEN
	fb_setpoint_switch_send.Group_Address.NUMBER:=REAL_TO_BYTE(dytjacha_hvac.cur_t_ust)+100;
	fb_setpoint_switch_send.Group_Address.MAIN:=1;
	fb_setpoint_switch_send.Group_Address.SUB_MAIN:=5;
	fb_setpoint_switch_send(str_Rec:=fb_KL6301_0.str_Data_Rec, bData:=1);
	fb_setpoint_switch_send(str_Rec:=fb_KL6301_0.str_Data_Rec, bData:=0);
END_IF
IF spalnya_hvac.cur_t_ust_prev <> spalnya_hvac.cur_t_ust THEN
	fb_setpoint_switch_send.Group_Address.NUMBER:=REAL_TO_BYTE(spalnya_hvac.cur_t_ust)+100;
	fb_setpoint_switch_send.Group_Address.MAIN:=1;
	fb_setpoint_switch_send.Group_Address.SUB_MAIN:=6;
	fb_setpoint_switch_send(str_Rec:=fb_KL6301_0.str_Data_Rec, bData:=1);
	fb_setpoint_switch_send(str_Rec:=fb_KL6301_0.str_Data_Rec, bData:=0);
END_IF
END_ACTION
ACTION timers:
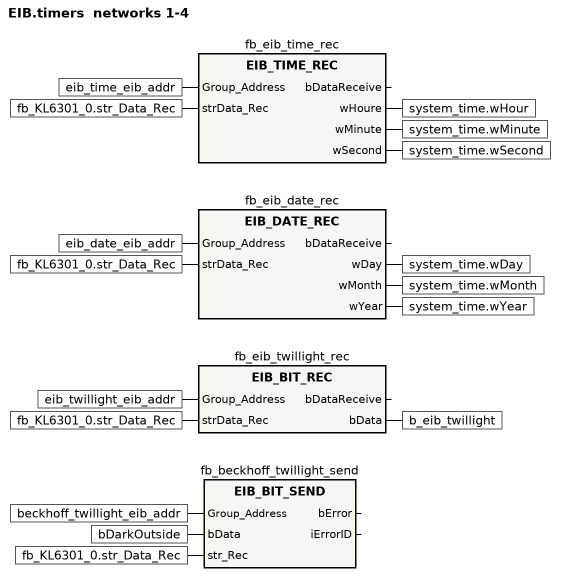
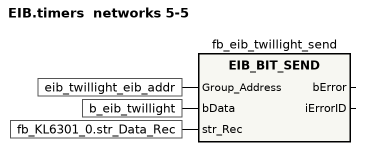
_FBD_ (* Function Block Diagram *)
NETWORK 1
	fb_eib_time_rec:EIB_TIME_REC(Group_Address: eib_time_eib_addr, strData_Rec: fb_KL6301_0.str_Data_Rec, wHoure => system_time.wHour, wMinute => system_time.wMinute, wSecond => system_time.wSecond)
NETWORK 2
	fb_eib_date_rec:EIB_DATE_REC(Group_Address: eib_date_eib_addr, strData_Rec: fb_KL6301_0.str_Data_Rec, wDay => system_time.wDay, wMonth => system_time.wMonth, wYear => system_time.wYear)
NETWORK 3
	fb_eib_twillight_rec:EIB_BIT_REC(Group_Address: eib_twillight_eib_addr, strData_Rec: fb_KL6301_0.str_Data_Rec, bData => b_eib_twillight)
NETWORK 4
	fb_beckhoff_twillight_send:EIB_BIT_SEND(Group_Address: beckhoff_twillight_eib_addr, bData: bDarkOutside, str_Rec: fb_KL6301_0.str_Data_Rec)
NETWORK 5
	fb_eib_twillight_send:EIB_BIT_SEND(Group_Address: eib_twillight_eib_addr, bData: b_eib_twillight, str_Rec: fb_KL6301_0.str_Data_Rec)
_END_FBD_
(* the same logic as Structured Text *)
(* Network 1 *)
fb_eib_time_rec(Group_Address := eib_time_eib_addr, strData_Rec := fb_KL6301_0.str_Data_Rec);
system_time.wHour := fb_eib_time_rec.wHoure;
system_time.wMinute := fb_eib_time_rec.wMinute;
system_time.wSecond := fb_eib_time_rec.wSecond;
(* Network 2 *)
fb_eib_date_rec(Group_Address := eib_date_eib_addr, strData_Rec := fb_KL6301_0.str_Data_Rec);
system_time.wDay := fb_eib_date_rec.wDay;
system_time.wMonth := fb_eib_date_rec.wMonth;
system_time.wYear := fb_eib_date_rec.wYear;
(* Network 3 *)
fb_eib_twillight_rec(Group_Address := eib_twillight_eib_addr, strData_Rec := fb_KL6301_0.str_Data_Rec);
b_eib_twillight := fb_eib_twillight_rec.bData;
(* Network 4 *)
fb_beckhoff_twillight_send(Group_Address := beckhoff_twillight_eib_addr, bData := bDarkOutside, str_Rec := fb_KL6301_0.str_Data_Rec);
(* Network 5 *)
fb_eib_twillight_send(Group_Address := eib_twillight_eib_addr, bData := b_eib_twillight, str_Rec := fb_KL6301_0.str_Data_Rec);
END_ACTION

(* POU HVAC/heat, ST *)
PROGRAM heat
VAR PERSISTENT

	t_out, t_out_avg_day, t_out_avg_10day:REAL;
	measures_this_day, meashured_days:INT;
	day_sum, ten_day_sum:REAL;
END_VAR


VAR
	temp_measure:TOF; (*таймер задає частоту замірів температури*)
	(*актуальна та попередня температури*)
	t_tambur, t_tamburPrev: REAL;
	t_su, t_suPrev: REAL;
	t_spalnya, t_spalnyaPrev: REAL;
	t_outPrev:REAL;
	(*мінімум та максимум температур теплих підлог*)
	t_max: REAL;
	t_min: REAL;
	(*різниця між поперднім та актуальним значенням температури*)
	delta_out, delta_tambur, delta_su, delta_spalnya: REAL;

	i: INT:=0;
	fbRetryCounter:CTU;
	iRetryCounter:INT;
	(*використовуються для знаходження середньої температури при ініціації*)
	t_tambur_sum: REAL;
	t_su_sum: REAL;
	t_spalnya_sum: REAL;
	t_out_sum: REAL;
	retry: BOOL:=TRUE;		(*переміряти температуру*)
END_VAR
(*фільтр показань сенсорів температури*)
CASE i OF
0..500: init;
ELSE
	IF retry THEN
		temp_measure.PT:=t#2s;

	ELSE temp_measure.PT:=t#5m;
	END_IF
	IF retry THEN
		IF iRetryCounter >5 THEN iRetryCounter:=0; i:=0; ELSE iRetryCounter:=iRetryCounter+1; END_IF;
	END_IF;
	temp_measure( IN:=NOT temp_measure.q); (*перевіряти температуру кожні 20 хв*)


IF NOT temp_measure.Q THEN

	delta_spalnya:=ABS(t_spalnyaPrev-temp_spalnya*0.1);
	delta_su:=ABS(t_suPrev-temp_su*0.1);
	delta_tambur:=ABS(t_tamburPrev-temp_tambur*0.1);
	delta_out:=ABS(t_outPrev-iT_out*0.1);
	retry:=FALSE;
	IF delta_spalnya<1 THEN
		t_spalnya:= temp_spalnya * 0.1;
	ELSE
		t_spalnya:=t_spalnyaPrev;
		retry:=TRUE;
	END_IF

	IF delta_su<1 THEN
		t_su:= temp_su * 0.1;
	ELSE
		t_su:=t_suPrev;
		retry:=TRUE;
	END_IF

	IF delta_tambur<1 THEN
		t_tambur:= temp_tambur * 0.1;
	ELSE
		t_tambur:=t_tamburPrev;
		retry:=TRUE;
	END_IF

	IF delta_out<01 THEN
		t_out:= iT_out* 0.1;
	ELSE
		t_out:=t_outPrev;
		retry:=TRUE;
	END_IF

	t_spalnyaPrev:=t_spalnya;
	t_suPrev:=t_su;
	t_tamburPrev:=t_tambur;
	t_outPrev:=t_out;

END_IF
END_CASE

(*CASE MAIN.fbRTC.stSystemTime.wSecond OF*)

IF t_out<0 THEN data1floor[2].7:=1; ELSE data1floor[2].7:=0; END_IF
data1floor[3]:=ABS(REAL_TO_BYTE(t_out));
data2floor[8]:=ABS(REAL_TO_BYTE(t_out));

(*summer; *)

t_max:=70;
t_min:=20;
IF t_out<15 THEN

	IF t_tambur > t_max THEN (*вимкнути колектор, якщо підлога тепліша за верхню межу температури*)
		freshbar_col:=FALSE;
	ELSE
		IF t_tambur< t_min THEN (*увімкнути колектор, якщо підлога холодніша за нижню межу*)
			freshbar_col:=TRUE;
		ELSE
			freshbar_col:= FALSE; (*ПОСТАВИТИ В ЗАЛЕЖНІСТЬ ВІД ЗОВНІШНЬОЇ ТЕМПЕРАТУРИ*)
		END_IF
	END_IF

	IF t_su > t_max THEN
		su_col_pidloga:=FALSE;
		su_col_stina:=FALSE;
			serverna_col:=FALSE;
	ELSE
		IF t_su< t_min THEN
			su_col_pidloga:=TRUE;
			su_col_stina:=TRUE;
			serverna_col:=TRUE;
		ELSE
			su_col_pidloga:=FALSE; (*ПОСТАВИТИ В ЗАЛЕЖНІСТЬ ВІД ЗОВНІШНЬОЇ ТЕМПЕРАТУРИ*)
			su_col_stina:=FALSE;
			serverna_col:=FALSE;
		END_IF
	END_IF

	IF t_spalnya>t_max THEN (*щоб не вистигала підлога*)
		spalnya_col:=FALSE;
	ELSE
		IF t_spalnya<t_min THEN
			spalnya_col:=TRUE;
		ELSE
			spalnya_col:=SPALNYA_HVAC.tepla_pidloga;
		END_IF
	END_IF


END_IF

(*

IF VITALNYA_HVAC.heat_mode=0 THEN
				VITALNYA_HVAC.fancoil_speed:=0;
				(*VITALNYA_HVAC.collector:=2#00000000; all closed*)
				VITALNYA_HVAC.klapan:=16#7FFF;(*full closed*)
				VITALNYA_HVAC.zaslinka:=TRUE;(*closed*)
	END_IF

	IF KINO_HVAC.heat_mode=0 THEN
				KINO_HVAC.fancoil_speed:=0;
				(*KINO_HVAC.collector:=2#00000000; all closed*)
				KINO_HVAC.klapan:=16#7FFF;(*full closed*)
				KINO_HVAC.zaslinka:=TRUE;(*closed*)
	END_IF

	IF STUDIO_HVAC.heat_mode=0 THEN
				STUDIO_HVAC.fancoil_speed:=0;
				(*STUDIO_HVAC.collector:=2#00000000; all closed*)
				STUDIO_HVAC.klapan:=16#7FFF;(*full closed*)
				STUDIO_HVAC.zaslinka:=TRUE;(*closed*)
	END_IF

	IF KABINET_HVAC.heat_mode=0 THEN
				KABINET_HVAC.fancoil_speed:=0;
				(*KABINET_HVAC.collector:=2#00000000; all closed*)
				KABINET_HVAC.klapan:=16#7FFF;(*full closed*)
				KABINET_HVAC.zaslinka:=TRUE;(*closed*)
	END_IF

	IF DYTJACHA_HVAC.heat_mode=0 THEN
				DYTJACHA_HVAC.fancoil_speed:=0;
				(*DYTJACHA_HVAC.collector:=2#00000000; all closed*)
				DYTJACHA_HVAC.klapan:=16#7FFF;(*full closed*)
				DYTJACHA_HVAC.zaslinka:=TRUE;(*closed*)
	END_IF

	IF SPALNYA_HVAC.heat_mode=0 THEN
				SPALNYA_HVAC.fancoil_speed:=0;
				(*SPALNYA_HVAC.collector:=2#00000000; all closed*)
				SPALNYA_HVAC.klapan:=16#7FFF;(*full closed*)
				SPALNYA_HVAC.zaslinka:=TRUE;(*closed*)
	END_IF
*)


data1floor[3]:=REAL_TO_BYTE (t_out);
data2floor[8]:=REAL_TO_BYTE (t_out);
data_derevo[3]:=REAL_TO_BYTE (t_out);
(*локальні змінні для фенкойлів 3го поверхну об'явлені в області виходів*)

(*------------------------fancoil speed --------------------------------------------------*)
IF EIB.fb_vitalnya_damper_ctrl_rec.bData THEN
	vitalnya_hvac.fancoil_speed:=1;
ELSE
	IF vitalnya_HVAC.heating_signal = 0  THEN
		CASE vitalnya_hvac.fancoil_speed OF
			0:	IF vitalnya_hvac.cooling_signal>0 THEN vitalnya_HVAC.fancoil_speed:=1; END_IF

			1:	IF vitalnya_hvac.cooling_signal=0 THEN vitalnya_HVAC.fancoil_speed:=0; END_IF
				IF vitalnya_hvac.cooling_signal>50 THEN  vitalnya_HVAC.fancoil_speed:=2; END_IF

			2:	IF vitalnya_hvac.cooling_signal=0 THEN vitalnya_HVAC.fancoil_speed:=0; END_IF
				IF vitalnya_hvac.cooling_signal>75  THEN vitalnya_HVAC.fancoil_speed:=3; END_IF
				IF vitalnya_hvac.cooling_signal<45  THEN vitalnya_HVAC.fancoil_speed:=1; END_IF

			3:	IF vitalnya_hvac.cooling_signal=0 THEN vitalnya_HVAC.fancoil_speed:=0; END_IF
				IF vitalnya_hvac.cooling_signal<75  THEN vitalnya_HVAC.fancoil_speed:=2; END_IF
		END_CASE
	END_IF

	IF vitalnya_HVAC.cooling_signal = 0 THEN
		CASE vitalnya_hvac.fancoil_speed OF
			0:	IF vitalnya_hvac.heating_signal>0 THEN vitalnya_HVAC.fancoil_speed:=1; END_IF

			1:	IF vitalnya_hvac.heating_signal=0 THEN vitalnya_HVAC.fancoil_speed:=0; END_IF
				IF vitalnya_hvac.heating_signal>50 THEN  vitalnya_HVAC.fancoil_speed:=2; END_IF

			2:	IF vitalnya_hvac.heating_signal=0 THEN vitalnya_HVAC.fancoil_speed:=0; END_IF
				IF vitalnya_hvac.heating_signal>75  THEN vitalnya_HVAC.fancoil_speed:=3; END_IF
				IF vitalnya_hvac.heating_signal<45  THEN vitalnya_HVAC.fancoil_speed:=1; END_IF

			3:	IF vitalnya_hvac.heating_signal=0 THEN vitalnya_HVAC.fancoil_speed:=0; END_IF
				IF vitalnya_hvac.heating_signal<75  THEN vitalnya_HVAC.fancoil_speed:=2; END_IF
		END_CASE
	END_IF
END_IF

IF EIB.fb_kino_damper_ctrl_rec.bData THEN
	kino_hvac.fancoil_speed:=1;
ELSE
	IF kino_HVAC.heating_signal = 0 THEN
		CASE kino_hvac.fancoil_speed OF
			0:	IF kino_hvac.cooling_signal>0 THEN kino_HVAC.fancoil_speed:=1; END_IF

			1:	IF kino_hvac.cooling_signal=0 THEN kino_HVAC.fancoil_speed:=0; END_IF
				IF kino_hvac.cooling_signal>50 THEN  kino_HVAC.fancoil_speed:=2; END_IF

			2:	IF kino_hvac.cooling_signal=0 THEN kino_HVAC.fancoil_speed:=0; END_IF
				IF kino_hvac.cooling_signal>75  THEN kino_HVAC.fancoil_speed:=3; END_IF
				IF kino_hvac.cooling_signal<45  THEN kino_HVAC.fancoil_speed:=1; END_IF

			3:	IF kino_hvac.cooling_signal=0 THEN kino_HVAC.fancoil_speed:=0; END_IF
				IF kino_hvac.cooling_signal<75  THEN kino_HVAC.fancoil_speed:=2; END_IF
		END_CASE
	END_IF
	IF kino_HVAC.cooling_signal = 0 THEN
		CASE kino_hvac.fancoil_speed OF
			0:	IF kino_hvac.heating_signal>0 THEN kino_HVAC.fancoil_speed:=1; END_IF

			1:	IF kino_hvac.heating_signal=0 THEN kino_HVAC.fancoil_speed:=0; END_IF
				IF kino_hvac.heating_signal>50 THEN  kino_HVAC.fancoil_speed:=2; END_IF

			2:	IF kino_hvac.heating_signal=0 THEN kino_HVAC.fancoil_speed:=0; END_IF
				IF kino_hvac.heating_signal>75  THEN kino_HVAC.fancoil_speed:=3; END_IF
				IF kino_hvac.heating_signal<45  THEN kino_HVAC.fancoil_speed:=1; END_IF

			3:	IF kino_hvac.heating_signal=0 THEN kino_HVAC.fancoil_speed:=0; END_IF
				IF kino_hvac.heating_signal<75  THEN kino_HVAC.fancoil_speed:=2; END_IF
		END_CASE
	END_IF
END_IF

IF EIB.fb_kabinet_damper_ctrl_rec.bData THEN
	kabinet_hvac.fancoil_speed:=1;
ELSE
	IF kabinet_HVAC.heating_signal = 0 THEN
		CASE kabinet_hvac.fancoil_speed OF
			0:	IF kabinet_hvac.cooling_signal>0 THEN kabinet_HVAC.fancoil_speed:=1; END_IF

			1:	IF kabinet_hvac.cooling_signal=0 THEN kabinet_HVAC.fancoil_speed:=0; END_IF
				IF kabinet_hvac.cooling_signal>50 THEN  kabinet_HVAC.fancoil_speed:=2; END_IF

			2:	IF kabinet_hvac.cooling_signal=0 THEN kabinet_HVAC.fancoil_speed:=0; END_IF
				IF kabinet_hvac.cooling_signal>75  THEN kabinet_HVAC.fancoil_speed:=3; END_IF
				IF kabinet_hvac.cooling_signal<45  THEN kabinet_HVAC.fancoil_speed:=1; END_IF

			3:	IF kabinet_hvac.cooling_signal=0 THEN kabinet_HVAC.fancoil_speed:=0; END_IF
				IF kabinet_hvac.cooling_signal<75  THEN kabinet_HVAC.fancoil_speed:=2; END_IF
		END_CASE
	END_IF
	IF kabinet_HVAC.cooling_signal = 0 THEN
		CASE kabinet_hvac.fancoil_speed OF
			0:	IF kabinet_hvac.heating_signal>0 THEN kabinet_HVAC.fancoil_speed:=1; END_IF

			1:	IF kabinet_hvac.heating_signal=0 THEN kabinet_HVAC.fancoil_speed:=0; END_IF
				IF kabinet_hvac.heating_signal>50 THEN  kabinet_HVAC.fancoil_speed:=2; END_IF

			2:	IF kabinet_hvac.heating_signal=0 THEN kabinet_HVAC.fancoil_speed:=0; END_IF
				IF kabinet_hvac.heating_signal>75  THEN kabinet_HVAC.fancoil_speed:=3; END_IF
				IF kabinet_hvac.heating_signal<45  THEN kabinet_HVAC.fancoil_speed:=1; END_IF

			3:	IF kabinet_hvac.heating_signal=0 THEN kabinet_HVAC.fancoil_speed:=0; END_IF
				IF kabinet_hvac.heating_signal<75  THEN kabinet_HVAC.fancoil_speed:=2; END_IF
		END_CASE
	END_IF
END_IF

IF EIB.fb_dytjacha_damper_ctrl_rec.bData THEN
	dytjacha_hvac.fancoil_speed:=1;
ELSE
	IF dytjacha_HVAC.heating_signal = 0 THEN
		CASE dytjacha_hvac.fancoil_speed OF
			0:	IF dytjacha_hvac.cooling_signal>0 THEN dytjacha_HVAC.fancoil_speed:=1; END_IF

			1:	IF dytjacha_hvac.cooling_signal=0 THEN dytjacha_HVAC.fancoil_speed:=0; END_IF
				IF dytjacha_hvac.cooling_signal>50 THEN  dytjacha_HVAC.fancoil_speed:=2; END_IF

			2:	IF dytjacha_hvac.cooling_signal=0 THEN dytjacha_HVAC.fancoil_speed:=0; END_IF
				IF dytjacha_hvac.cooling_signal>75  THEN dytjacha_HVAC.fancoil_speed:=3; END_IF
				IF dytjacha_hvac.cooling_signal<45  THEN dytjacha_HVAC.fancoil_speed:=1; END_IF

			3:	IF dytjacha_hvac.cooling_signal=0 THEN dytjacha_HVAC.fancoil_speed:=0; END_IF
				IF dytjacha_hvac.cooling_signal<75  THEN dytjacha_HVAC.fancoil_speed:=2; END_IF
		END_CASE
	END_IF
	IF dytjacha_HVAC.cooling_signal = 0 THEN
		CASE dytjacha_hvac.fancoil_speed OF
			0:	IF dytjacha_hvac.heating_signal>0 THEN dytjacha_HVAC.fancoil_speed:=1; END_IF

			1:	IF dytjacha_hvac.heating_signal=0 THEN dytjacha_HVAC.fancoil_speed:=0; END_IF
				IF dytjacha_hvac.heating_signal>50 THEN  dytjacha_HVAC.fancoil_speed:=2; END_IF

			2:	IF dytjacha_hvac.heating_signal=0 THEN dytjacha_HVAC.fancoil_speed:=0; END_IF
				IF dytjacha_hvac.heating_signal>75  THEN dytjacha_HVAC.fancoil_speed:=3; END_IF
				IF dytjacha_hvac.heating_signal<45  THEN dytjacha_HVAC.fancoil_speed:=1; END_IF

			3:	IF dytjacha_hvac.heating_signal=0 THEN dytjacha_HVAC.fancoil_speed:=0; END_IF
				IF dytjacha_hvac.heating_signal<75  THEN dytjacha_HVAC.fancoil_speed:=2; END_IF
		END_CASE
	END_IF
END_IF

IF EIB.fb_spalnya_damper_ctrl_rec.bData THEN
	spalnya_hvac.fancoil_speed:=1;
ELSE
	IF spalnya_HVAC.heating_signal = 0 THEN
		CASE spalnya_hvac.fancoil_speed OF
			0:	IF spalnya_hvac.cooling_signal>0 THEN spalnya_HVAC.fancoil_speed:=1; END_IF

			1:	IF spalnya_hvac.cooling_signal=0 THEN spalnya_HVAC.fancoil_speed:=0; END_IF
				IF spalnya_hvac.cooling_signal>50 THEN  spalnya_HVAC.fancoil_speed:=2; END_IF

			2:	IF spalnya_hvac.cooling_signal=0 THEN spalnya_HVAC.fancoil_speed:=0; END_IF
				IF spalnya_hvac.cooling_signal>75  THEN spalnya_HVAC.fancoil_speed:=3; END_IF
				IF spalnya_hvac.cooling_signal<45  THEN spalnya_HVAC.fancoil_speed:=1; END_IF

			3:	IF spalnya_hvac.cooling_signal=0 THEN spalnya_HVAC.fancoil_speed:=0; END_IF
				IF spalnya_hvac.cooling_signal<75  THEN spalnya_HVAC.fancoil_speed:=2; END_IF
		END_CASE
	END_IF
	IF spalnya_HVAC.cooling_signal = 0 THEN
		CASE spalnya_hvac.fancoil_speed OF
			0:	IF spalnya_hvac.heating_signal>0 THEN spalnya_HVAC.fancoil_speed:=1; END_IF

			1:	IF spalnya_hvac.heating_signal=0 THEN spalnya_HVAC.fancoil_speed:=0; END_IF
				IF spalnya_hvac.heating_signal>50 THEN  spalnya_HVAC.fancoil_speed:=2; END_IF

			2:	IF spalnya_hvac.heating_signal=0 THEN spalnya_HVAC.fancoil_speed:=0; END_IF
				IF spalnya_hvac.heating_signal>75  THEN spalnya_HVAC.fancoil_speed:=3; END_IF
				IF spalnya_hvac.heating_signal<45  THEN spalnya_HVAC.fancoil_speed:=1; END_IF

			3:	IF spalnya_hvac.heating_signal=0 THEN spalnya_HVAC.fancoil_speed:=0; END_IF
				IF spalnya_hvac.heating_signal<75  THEN spalnya_HVAC.fancoil_speed:=2; END_IF
		END_CASE
	END_IF
END_IF
CASE DYTJACHA_HVAC.fancoil_speed OF
	0:	fancoil_dytjacha_low:=FALSE;
		fancoil_dytjacha_med:=FALSE;
		fancoil_dytjacha_high:=FALSE;

	1:	fancoil_dytjacha_low:=TRUE;
		fancoil_dytjacha_med:=FALSE;
		fancoil_dytjacha_high:=FALSE;

	2:	fancoil_dytjacha_low:=FALSE;
		fancoil_dytjacha_med:=TRUE;
		fancoil_dytjacha_high:=FALSE;

	3:	fancoil_dytjacha_low:=FALSE;
		fancoil_dytjacha_med:=FALSE;
		fancoil_dytjacha_high:=TRUE;
END_CASE

CASE SPALNYA_HVAC.fancoil_speed OF
	0:	fancoil_spalnya_low:=FALSE;
		fancoil_spalnya_med:=FALSE;
		fancoil_spalnya_high:=FALSE;

	1:	fancoil_spalnya_low:=TRUE;
		fancoil_spalnya_med:=FALSE;
		fancoil_spalnya_high:=FALSE;

	2:	fancoil_spalnya_low:=FALSE;
		fancoil_spalnya_med:=TRUE;
		fancoil_spalnya_high:=FALSE;

	3:	fancoil_spalnya_low:=FALSE;
		fancoil_spalnya_med:=FALSE;
		fancoil_spalnya_high:=TRUE;
END_CASE
CASE KABINET_HVAC.fancoil_speed OF
	0:	data2floor[0].0:=0; (*запис в масив даних, що відправляються на 2й поверх*)
		data2floor[0].1:=0;
		data2floor[0].2:=0;

	1:	data2floor[0].0:=1; (*запис в масив даних, що відправляються на 2й поверх*)
		data2floor[0].1:=0;
		data2floor[0].2:=0;

	2:	data2floor[0].0:=0; (*запис в масив даних, що відправляються на 2й поверх*)
		data2floor[0].1:=1;
		data2floor[0].2:=0;

	3:	data2floor[0].0:=0; (*запис в масив даних, що відправляються на 2й поверх*)
		data2floor[0].1:=0;
		data2floor[0].2:=1;
END_CASE

CASE KINO_HVAC.fancoil_speed OF
	0:	data2floor[0].3:=0; (*запис в масив даних, що відправляються на 2й поверх*)
		data2floor[0].4:=0;
		data2floor[0].5:=0;

	1:	data2floor[0].3:=1; (*запис в масив даних, що відправляються на 2й поверх*)
		data2floor[0].4:=0;
		data2floor[0].5:=0;

	2:	data2floor[0].3:=0; (*запис в масив даних, що відправляються на 2й поверх*)
		data2floor[0].4:=1;
		data2floor[0].5:=0;

	3:	data2floor[0].3:=0; (*запис в масив даних, що відправляються на 2й поверх*)
		data2floor[0].4:=0;
		data2floor[0].5:=1;
END_CASE

CASE VITALNYA_HVAC.fancoil_speed OF
	0:	data1floor[0].0:=0; (*запис в масив даних, що відправляються на 1й поверх*)
		data1floor[0].1:=0;
		data1floor[0].2:=0;

	1:	data1floor[0].0:=1; (*запис в масив даних, що відправляються на 1й поверх*)
		data1floor[0].1:=0;
		data1floor[0].2:=0;

	2:	data1floor[0].0:=0; (*запис в масив даних, що відправляються на 1й поверх*)
		data1floor[0].1:=1;
		data1floor[0].2:=0;

	3:	data1floor[0].0:=0; (*запис в масив даних, що відправляються на 1й поверх*)
		data1floor[0].1:=0;
		data1floor[0].2:=1;
END_CASE

(*--------------------------------------klapany--------------------------------------------*)
(*data1floor[2]:=WORD_TO_BYTE(VITALNYA_HVAC.klapan); data1floor[3]:=WORD_TO_BYTE(SHR(VITALNYA_HVAC.klapan,8));*)
klapan_vitalnya:=VITALNYA_HVAC.klapan;
klapan_spalnya:=SPALNYA_HVAC.klapan;
klapan_dytjacha:=DYTJACHA_HVAC.klapan;

data2floor[2]:=WORD_TO_BYTE(KABINET_HVAC.klapan); data2floor[3]:=WORD_TO_BYTE(SHR(KABINET_HVAC.klapan,8));
data2floor[4]:=WORD_TO_BYTE(KINO_HVAC.klapan); data2floor[5]:=WORD_TO_BYTE(SHR(KINO_HVAC.klapan,8));

(*------------------------------zaslinky------------------------------------*)
z_vitalnya:=VITALNYA_HVAC.zaslinka;
z_kabinet:=KABINET_HVAC.zaslinka;
z_kino:=KINO_HVAC.zaslinka;
z_dytjacha:=DYTJACHA_HVAC.zaslinka;
z_spalnya:=SPALNYA_HVAC.zaslinka;

(*-----------------------------tepla pidloga-------------------------------*)
data1floor[0].4:=VITALNYA_HVAC.tepla_pidloga;
data2floor[1].0:=KABINET_HVAC.tepla_pidloga;
data2floor[1].1:=KABINET_HVAC.tepla_pidloga;
data2floor[1].2:=STUDIO_HVAC.tepla_pidloga;
data2floor[1].3:=STUDIO_HVAC.tepla_pidloga;

dytjacha_col:=DYTJACHA_HVAC.tepla_pidloga;
spalnya_col:=SPALNYA_HVAC.tepla_pidloga;
END_PROGRAM
ACTION init:
IF i=500 THEN
	t_tamburPrev:=t_tambur_sum/i;
	t_suPrev:=t_su_sum/i;
	t_spalnyaPrev:=t_spalnya_sum/i;
	t_outPrev:=t_out_sum/i;
	t_tambur_sum:=0;
	t_su_sum:=0;
	t_spalnya_sum:=0;
	t_out_sum:=0;
	i:=501;
ELSE
	t_tambur_sum:=t_tambur_sum+temp_tambur*0.1;
	t_su_sum:=t_su_sum+temp_su*0.1;
	t_spalnya_sum:=t_spalnya_sum+temp_spalnya*0.1;
	t_out_sum:=t_out_sum+iT_out*0.1;
	i:=i+1;
END_IF
END_ACTION

(* POU ADS_write, ST *)
PROGRAM ADS_write
VAR
	write_timeout: TIME;
	b_write1, b_write2: BOOL;
	write_ads1, write_ads2, write_ads4: ADSWRITE;

	timer1, timer2:TP;
	errorcounter1, errorcounter2, pack_c:CTU ;
	test_word: WORD;
	i,j,i1,j1, i4,j4: INT;
	data_changed: BOOL;
	try_again2, try_again1, try_again4: BOOL;
	timer4: TP;
	b_write4: BOOL;
	errorcounter4: CTU;
END_VAR
write_timeout:=t#3s;

FOR i:=0 TO (SIZEOF(data2floor))-1 DO
	IF data2floor[i]<>data2floor_prev[i]  OR try_again2 THEN
		b_write2:=TRUE;
		EXIT;
	ELSE
		b_write2:=FALSE;
	END_IF
END_FOR

IF write_ads2.BUSY THEN b_write2:=FALSE; END_IF

	write_ads2(
		NETID:=ads_adr2,
		PORT:=800,
		IDXGRP:=16#4020,
		IDXOFFS:=300,
		WRITE:=b_write2,
		TMOUT:=write_timeout,
		LEN:=SIZEOF(data2floor),
		SRCADDR:=ADR(data2floor));
write_ads2.WRITE:=FALSE;

IF write_ads2.ERR AND NOT timer2.Q THEN
	timer2.IN:=TRUE;
	try_again2:=TRUE;
ELSE try_again2:=FALSE;
END_IF
timer2(PT:=write_timeout*2);
timer2.IN:=FALSE;


FOR j:=0 TO (SIZEOF(data2floor))-1 DO
	data2floor_prev[j]:=data2floor[j];
END_FOR

(*1floor*)
FOR i1:=0 TO (SIZEOF(data1floor))-1 DO
	IF data1floor[i1]<>data1floor_prev[i1] AND NOT timer1.Q THEN
		b_write1:=TRUE;
		EXIT;
	ELSE
		b_write1:=FALSE;
	END_IF
END_FOR

IF try_again1 AND NOT timer1.Q THEN
	b_write1:=TRUE;
	try_again1:=FALSE;
END_IF

errorcounter1(cu:=write_ads1.ERR);


IF write_ads1.BUSY THEN b_write1:=FALSE; END_IF

	write_ads1(
		NETID:=ads_adr1,
		PORT:=800,
		IDXGRP:=16#4020,
		IDXOFFS:=300,
		WRITE:=b_write1,
		TMOUT:=write_timeout,
		LEN:=SIZEOF(data1floor),
		SRCADDR:=ADR(data1floor));

IF write_ads1.ERR AND NOT timer1.Q THEN
	timer1.IN:=TRUE;
	try_again1:=TRUE;
END_IF
timer1(PT:=write_timeout);
timer1.IN:=FALSE;


FOR j1:=0 TO (SIZEOF(data1floor))-1 DO
	data1floor_prev[j1]:=data1floor[j1];
END_FOR

(*derevo*)
FOR i4:=0 TO (SIZEOF(data_derevo))-1 DO
	IF data_derevo[i4]<>data_derevo_prev[i4] AND NOT timer4.Q THEN
		b_write4:=TRUE;
		EXIT;
	ELSE
		b_write4:=FALSE;
	END_IF
END_FOR

IF try_again4 AND NOT timer4.Q THEN
	b_write4:=TRUE;
	try_again4:=FALSE;
END_IF

errorcounter4(cu:=write_ads4.ERR);


IF write_ads4.BUSY THEN b_write4:=FALSE; END_IF

	write_ads4(
		NETID:=ads_adr4,
		PORT:=800,
		IDXGRP:=16#4020,
		IDXOFFS:=400,
		WRITE:=b_write4,
		TMOUT:=write_timeout,
		LEN:=SIZEOF(data_derevo),
		SRCADDR:=ADR(data_derevo));

IF write_ads4.ERR AND NOT timer4.Q THEN
	timer4.IN:=TRUE;
	try_again4:=TRUE;
END_IF
timer4(PT:=write_timeout);
timer4.IN:=FALSE;


FOR j4:=0 TO (SIZEOF(data_derevo))-1 DO
	data_derevo_prev[j4]:=data_derevo[j4];
END_FOR
END_PROGRAM

(* POU RANGE_TO_RANGE, ST *)
FUNCTION RANGE_TO_RANGE : INT
VAR_INPUT
	by_input:BYTE;
	in_low_value: INT;
	in_high_value:INT;
	out_low_value: INT;
	out_high_value:INT;
END_VAR
VAR
	r_res: REAL;
	r_input: REAL;
END_VAR
r_input:=BYTE_TO_REAL(by_input);
IF out_high_value>out_low_value THEN
	r_res:=r_input/(in_high_value - in_low_value)*(out_high_value - out_low_value);
ELSE
	r_res:=out_low_value - (r_input / (in_high_value - in_low_value)*(out_low_value - out_high_value));
END_IF
RANGE_TO_RANGE:=REAL_TO_INT(r_res);
END_FUNCTION

(* POU GREATEST_OF, ST *)
FUNCTION GREATEST_OF : REAL
VAR_INPUT
	r_in1,r_in2:REAL;
END_VAR
VAR
END_VAR
IF r_in1>=r_in2 THEN
	GREATEST_OF:=r_in1;
ELSE
	GREATEST_OF:=r_in2;
END_IF
END_FUNCTION

(* POU LIGHT_cfc, CFC *)
PROGRAM LIGHT_cfc
VAR
	tamburSw1: FB_ShortLongClick;
	tamburSw2: FB_ShortLongClick;
	tamburSw3: FB_ShortLongClick;
	spalnyaSw1: FB_ShortLongClick;
	spalnyaSw2: FB_ShortLongClick;
	spalnyaBalcSw: FB_ShortLongClick;
	dytjachaSw1: FB_ShortLongClick;
	dytjachaSw2: FB_ShortLongClick;
	suSw1: FB_ShortLongClick;
	suSw2: FB_ShortLongClick;
	barLight: FB_Light;
END_VAR
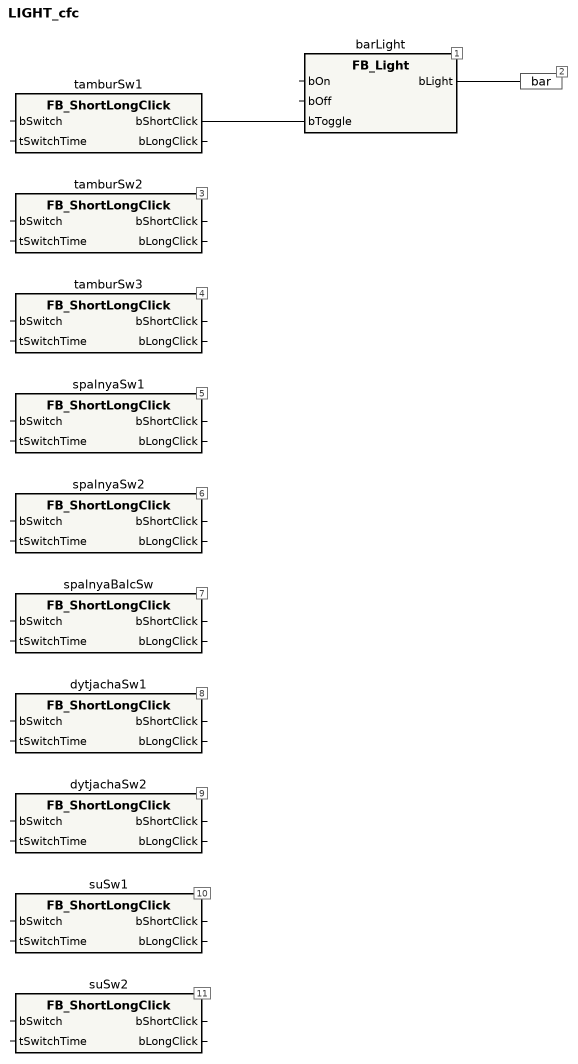
_CFC_ (* Continuous Function Chart, elements in execution order *)
#0 tamburSw1:FB_ShortLongClick(bSwitch: -, tSwitchTime: -)
#1 barLight:FB_Light(bOn: -, bOff: -, bToggle: #0.bShortClick)
#2 bar <= #1.bLight
#3 tamburSw2:FB_ShortLongClick(bSwitch: -, tSwitchTime: -)
#4 tamburSw3:FB_ShortLongClick(bSwitch: -, tSwitchTime: -)
#5 spalnyaSw1:FB_ShortLongClick(bSwitch: -, tSwitchTime: -)
#6 spalnyaSw2:FB_ShortLongClick(bSwitch: -, tSwitchTime: -)
#7 spalnyaBalcSw:FB_ShortLongClick(bSwitch: -, tSwitchTime: -)
#8 dytjachaSw1:FB_ShortLongClick(bSwitch: -, tSwitchTime: -)
#9 dytjachaSw2:FB_ShortLongClick(bSwitch: -, tSwitchTime: -)
#10 suSw1:FB_ShortLongClick(bSwitch: -, tSwitchTime: -)
#11 suSw2:FB_ShortLongClick(bSwitch: -, tSwitchTime: -)
_END_CFC_
(* the same logic as Structured Text *)
tamburSw1();
barLight(bToggle := tamburSw1.bShortClick);
bar := barLight.bLight;
tamburSw2();
tamburSw3();
spalnyaSw1();
spalnyaSw2();
spalnyaBalcSw();
dytjachaSw1();
dytjachaSw2();
suSw1();
suSw2();
END_PROGRAM

(* POU HVAC/summer, ST *)
PROGRAM summer
VAR

END_VAR
data1floor[0].3:=heating_mode;

(*--------------------------VITALNYA---------------------------------------------------------------*)

	IF VITALNYA_HVAC.heat_mode=2 THEN (*heat*)
		IF heating_mode THEN VITALNYA_HVAC.zaslinka:=TRUE;(*closed*) ELSE VITALNYA_HVAC.zaslinka:=FALSE; (*opened*)END_IF;
		VITALNYA_HVAC.tepla_pidloga:=TRUE; (*all opened*);
		CASE VITALNYA_HVAC.heat_speed OF
			1:	VITALNYA_HVAC.fancoil_speed:=1;
				IF NOT heating_mode THEN  VITALNYA_HVAC.klapan:=16#0; ELSE VITALNYA_HVAC.klapan:=16#3FFF;END_IF
			2:	VITALNYA_HVAC.fancoil_speed:=2;
				IF NOT heating_mode THEN  VITALNYA_HVAC.klapan:=16#0; ELSE VITALNYA_HVAC.klapan:=16#5FFF;END_IF
			3:	VITALNYA_HVAC.fancoil_speed:=3;
				IF NOT heating_mode THEN  VITALNYA_HVAC.klapan:=16#0; ELSE VITALNYA_HVAC.klapan:=16#7FFF;END_IF
		END_CASE
	END_IF

	IF VITALNYA_HVAC.heat_mode=1 THEN (*cool*)
		IF  heating_mode THEN VITALNYA_HVAC.klapan:=16#0;(*full closed*) END_IF
		IF  heating_mode THEN VITALNYA_HVAC.zaslinka:=FALSE; ELSE VITALNYA_HVAC.zaslinka:=TRUE; END_IF
				VITALNYA_HVAC.tepla_pidloga:=FALSE; (*all closed*)

			CASE VITALNYA_HVAC.heat_speed OF
			1:	VITALNYA_HVAC.fancoil_speed:=1;
				IF NOT heating_mode THEN  VITALNYA_HVAC.klapan:=16#3FFF; ELSE VITALNYA_HVAC.klapan:=16#0;END_IF
			2:	VITALNYA_HVAC.fancoil_speed:=2;
				IF NOT heating_mode THEN  VITALNYA_HVAC.klapan:=16#5FFF; ELSE VITALNYA_HVAC.klapan:=16#0;END_IF
			3:	VITALNYA_HVAC.fancoil_speed:=3;
				IF NOT heating_mode THEN  VITALNYA_HVAC.klapan:=16#7FFF; ELSE VITALNYA_HVAC.klapan:=16#0;END_IF
		END_CASE
	END_IF

	IF VITALNYA_HVAC.heat_mode=3 THEN (*fan*)
		VITALNYA_HVAC.tepla_pidloga:=FALSE;

		CASE VITALNYA_HVAC.heat_speed OF
			1:	VITALNYA_HVAC.fancoil_speed:=0;
				VITALNYA_HVAC.zaslinka:=TRUE;(*closed*)
				VITALNYA_HVAC.klapan:=16#0;(*full closed*)
			2:	VITALNYA_HVAC.fancoil_speed:=2;
				VITALNYA_HVAC.zaslinka:=FALSE;(*opened*)
				VITALNYA_HVAC.klapan:=16#7FFF;
			3:	VITALNYA_HVAC.fancoil_speed:=3;
				VITALNYA_HVAC.zaslinka:=FALSE;(*opened*)
				VITALNYA_HVAC.klapan:=16#7FFF;
		END_CASE
	IF heat.t_out<0 THEN VITALNYA_HVAC.klapan:=16#5FFF; ELSE VITALNYA_HVAC.klapan:=16#0;END_IF
	END_IF



(*--------------------------KABINET---------------------------------------------------------------*)
(*реверс двигуна клапана*)

	IF kabinet_HVAC.heat_mode=2 THEN (*heat*)
		IF heating_mode THEN kabinet_HVAC.zaslinka:=TRUE;(*closed*) ELSE kabinet_HVAC.zaslinka:=FALSE; (*opened*)END_IF;
		kabinet_HVAC.tepla_pidloga:=TRUE; (*all opened*);
		CASE kabinet_HVAC.heat_speed OF
			1:	kabinet_HVAC.fancoil_speed:=1;
				IF heating_mode THEN  kabinet_HVAC.klapan:=16#0; ELSE kabinet_HVAC.klapan:=16#7FFF;END_IF
			2:	kabinet_HVAC.fancoil_speed:=2;
				IF heating_mode THEN  kabinet_HVAC.klapan:=16#0; ELSE kabinet_HVAC.klapan:=16#5FFF;END_IF
			3:	kabinet_HVAC.fancoil_speed:=3;
				IF heating_mode THEN  kabinet_HVAC.klapan:=16#0; ELSE kabinet_HVAC.klapan:=16#3FFF;END_IF
		END_CASE
	END_IF

	IF kabinet_HVAC.heat_mode=1 THEN (*cool*)
		IF NOT heating_mode THEN kabinet_HVAC.klapan:=16#0;(*full closed*) END_IF
		IF NOT heating_mode THEN kabinet_HVAC.zaslinka:=FALSE; ELSE kabinet_HVAC.zaslinka:=TRUE; END_IF
				kabinet_HVAC.tepla_pidloga:=FALSE; (*all closed*)

			CASE kabinet_HVAC.heat_speed OF
			1:	kabinet_HVAC.fancoil_speed:=1;
				IF heating_mode THEN  kabinet_HVAC.klapan:=16#7FFF; ELSE kabinet_HVAC.klapan:=16#0;END_IF
			2:	kabinet_HVAC.fancoil_speed:=2;
				IF heating_mode THEN  kabinet_HVAC.klapan:=16#5FFF; ELSE kabinet_HVAC.klapan:=16#0;END_IF
			3:	kabinet_HVAC.fancoil_speed:=3;
				IF heating_mode THEN  kabinet_HVAC.klapan:=16#3FFF; ELSE kabinet_HVAC.klapan:=16#0;END_IF
		END_CASE
	END_IF

	IF kabinet_HVAC.heat_mode=3 THEN (*fan*)
		kabinet_HVAC.tepla_pidloga:=FALSE;
		IF heat.t_out<0 THEN kabinet_HVAC.klapan:=16#3FFF;(*30%*) ELSE kabinet_HVAC.klapan:=16#0;END_IF
		CASE kabinet_HVAC.heat_speed OF
			1:	kabinet_HVAC.fancoil_speed:=0;
				kabinet_HVAC.zaslinka:=TRUE;(*closed*)
				kabinet_HVAC.klapan:=16#0;(*full closed*)
			2:	kabinet_HVAC.fancoil_speed:=2;
				kabinet_HVAC.zaslinka:=FALSE;(*opened*)
				kabinet_HVAC.klapan:=16#7FFF;
			3:	kabinet_HVAC.fancoil_speed:=3;
				kabinet_HVAC.zaslinka:=FALSE;(*opened*)
				kabinet_HVAC.klapan:=16#7FFF;
		END_CASE
	END_IF


(*--------------------------KINO---------------------------------------------------------------*)
(*реверс двигуна клапана*)

	IF KINO_HVAC.heat_mode=2 THEN (*heat*)
		IF heating_mode THEN KINO_HVAC.zaslinka:=TRUE;(*closed*) ELSE KINO_HVAC.zaslinka:=FALSE; (*opened*)END_IF;
		KINO_HVAC.tepla_pidloga:=TRUE; (*all opened*);
		CASE KINO_HVAC.heat_speed OF
			1:	KINO_HVAC.fancoil_speed:=1;
				IF NOT heating_mode THEN  KINO_HVAC.klapan:=16#0; ELSE KINO_HVAC.klapan:=16#5FFF;END_IF
			2:	KINO_HVAC.fancoil_speed:=2;
				IF NOT heating_mode THEN  KINO_HVAC.klapan:=16#0; ELSE KINO_HVAC.klapan:=16#3FFF;END_IF
			3:	KINO_HVAC.fancoil_speed:=3;
				IF NOT heating_mode THEN  KINO_HVAC.klapan:=16#0; ELSE KINO_HVAC.klapan:=16#0;END_IF
		END_CASE
	END_IF

	IF KINO_HVAC.heat_mode=1 THEN (*cool*)
		IF  heating_mode THEN KINO_HVAC.klapan:=16#7FFF;(*full closed*) END_IF
		IF  heating_mode THEN KINO_HVAC.zaslinka:=FALSE; ELSE KINO_HVAC.zaslinka:=TRUE; END_IF
				KINO_HVAC.tepla_pidloga:=FALSE; (*all closed*)

			CASE KINO_HVAC.heat_speed OF
			1:	KINO_HVAC.fancoil_speed:=1;
				IF NOT heating_mode THEN  KINO_HVAC.klapan:=16#5FFF; ELSE KINO_HVAC.klapan:=16#7FFF;END_IF
			2:	KINO_HVAC.fancoil_speed:=2;
				IF NOT heating_mode THEN  KINO_HVAC.klapan:=16#3FFF; ELSE KINO_HVAC.klapan:=16#7FFF;END_IF
			3:	KINO_HVAC.fancoil_speed:=3;
				IF NOT heating_mode THEN  KINO_HVAC.klapan:=16#0; ELSE KINO_HVAC.klapan:=16#7FFF;END_IF
		END_CASE
	END_IF

	IF KINO_HVAC.heat_mode=3 THEN (*fan*)
		KINO_HVAC.tepla_pidloga:=FALSE;

		CASE KINO_HVAC.heat_speed OF
			1:	KINO_HVAC.fancoil_speed:=0;
				KINO_HVAC.zaslinka:=TRUE;(*closed*)
				KINO_HVAC.klapan:=16#7FFF;(*full closed*)
			2:	KINO_HVAC.fancoil_speed:=2;
				KINO_HVAC.zaslinka:=FALSE;(*opened*)
				KINO_HVAC.klapan:=16#7FFF;
			3:	KINO_HVAC.fancoil_speed:=3;
				KINO_HVAC.zaslinka:=FALSE;(*opened*)
				KINO_HVAC.klapan:=16#7FFF;
		END_CASE
		IF heat.t_out<0 THEN KINO_HVAC.klapan:=16#5FFF;  ELSE KINO_HVAC.klapan:=16#7FFF;END_IF
	END_IF

(*--------------------------DYTJACHA---------------------------------------------------------------*)
(*реверс двигуна клапана*)

	IF dytjacha_HVAC.heat_mode=2 THEN (*heat*)
		IF heating_mode THEN dytjacha_HVAC.zaslinka:=TRUE;(*closed*) ELSE dytjacha_HVAC.zaslinka:=FALSE; (*opened*)END_IF;
		dytjacha_HVAC.tepla_pidloga:=TRUE; (*all opened*);
		CASE dytjacha_HVAC.heat_speed OF
			1:	dytjacha_HVAC.fancoil_speed:=1;
				IF NOT heating_mode THEN  dytjacha_HVAC.klapan:=16#7FFF; ELSE dytjacha_HVAC.klapan:=16#5FFF;END_IF
			2:	dytjacha_HVAC.fancoil_speed:=2;
				IF NOT heating_mode THEN  dytjacha_HVAC.klapan:=16#7FFF; ELSE dytjacha_HVAC.klapan:=16#3FFF;END_IF
			3:	dytjacha_HVAC.fancoil_speed:=3;
				IF NOT heating_mode THEN  dytjacha_HVAC.klapan:=16#7FFF; ELSE dytjacha_HVAC.klapan:=16#0;END_IF
		END_CASE
	END_IF

	IF dytjacha_HVAC.heat_mode=1 THEN (*cool*)
		IF  heating_mode THEN dytjacha_HVAC.klapan:=16#7FFF;(*full closed*) END_IF
		IF  heating_mode THEN dytjacha_HVAC.zaslinka:=FALSE; ELSE dytjacha_HVAC.zaslinka:=TRUE; END_IF
				dytjacha_HVAC.tepla_pidloga:=FALSE; (*all closed*)

			CASE dytjacha_HVAC.heat_speed OF
			1:	dytjacha_HVAC.fancoil_speed:=1;
				IF heating_mode THEN  dytjacha_HVAC.klapan:=16#7FFF; ELSE dytjacha_HVAC.klapan:=16#0;END_IF
			2:	dytjacha_HVAC.fancoil_speed:=2;
				IF heating_mode THEN  dytjacha_HVAC.klapan:=16#5FFF; ELSE dytjacha_HVAC.klapan:=16#0;END_IF
			3:	dytjacha_HVAC.fancoil_speed:=3;
				IF heating_mode THEN  dytjacha_HVAC.klapan:=16#3FFF; ELSE dytjacha_HVAC.klapan:=16#0;END_IF
		END_CASE
	END_IF

	IF dytjacha_HVAC.heat_mode=3 THEN (*fan*)
		dytjacha_HVAC.tepla_pidloga:=FALSE;
		CASE dytjacha_HVAC.heat_speed OF
			1:	dytjacha_HVAC.fancoil_speed:=0;
				dytjacha_HVAC.zaslinka:=TRUE;(*closed*)
				dytjacha_HVAC.klapan:=16#0;(*full closed*)
			2:	dytjacha_HVAC.fancoil_speed:=2;
				dytjacha_HVAC.zaslinka:=FALSE;(*opened*)
				dytjacha_HVAC.klapan:=16#7FFF;
			3:	dytjacha_HVAC.fancoil_speed:=3;
				dytjacha_HVAC.zaslinka:=FALSE;(*opened*)
				dytjacha_HVAC.klapan:=16#7FFF;
		END_CASE
		IF heat.t_out<0 THEN dytjacha_HVAC.klapan:=16#5FFF; ELSE dytjacha_HVAC.klapan:=16#7FFF;END_IF
	END_IF
(*--------------------------SPALNYA---------------------------------------------------------------*)

	IF SPALNYA_HVAC.heat_mode=2 THEN (*heat*)
		IF heating_mode THEN SPALNYA_HVAC.zaslinka:=TRUE;(*closed*) ELSE SPALNYA_HVAC.zaslinka:=FALSE; (*opened*)END_IF;
		SPALNYA_HVAC.tepla_pidloga:=TRUE; (*all opened*);
		CASE SPALNYA_HVAC.heat_speed OF
			1:	SPALNYA_HVAC.fancoil_speed:=1;
				IF NOT  heating_mode THEN  SPALNYA_HVAC.klapan:=16#0; ELSE SPALNYA_HVAC.klapan:=16#3FFF;END_IF
			2:	SPALNYA_HVAC.fancoil_speed:=2;
				IF NOT heating_mode THEN  SPALNYA_HVAC.klapan:=16#0; ELSE SPALNYA_HVAC.klapan:=16#5FFF;END_IF
			3:	SPALNYA_HVAC.fancoil_speed:=3;
				IF NOT heating_mode THEN  SPALNYA_HVAC.klapan:=16#0; ELSE SPALNYA_HVAC.klapan:=16#7FFF;END_IF
		END_CASE
	END_IF

	IF SPALNYA_HVAC.heat_mode=1 THEN (*cool*)
		IF  heating_mode THEN SPALNYA_HVAC.klapan:=16#5FFF;(*full closed*) END_IF
		IF  heating_mode THEN SPALNYA_HVAC.zaslinka:=FALSE; ELSE SPALNYA_HVAC.zaslinka:=TRUE; END_IF
				SPALNYA_HVAC.tepla_pidloga:=FALSE; (*all closed*)

			CASE SPALNYA_HVAC.heat_speed OF
			1:	SPALNYA_HVAC.fancoil_speed:=1;
				IF NOT heating_mode THEN  SPALNYA_HVAC.klapan:=16#3FFF; ELSE SPALNYA_HVAC.klapan:=16#0;END_IF
			2:	SPALNYA_HVAC.fancoil_speed:=2;
				IF NOT heating_mode THEN  SPALNYA_HVAC.klapan:=16#5FFF; ELSE SPALNYA_HVAC.klapan:=16#0;END_IF
			3:	SPALNYA_HVAC.fancoil_speed:=3;
				IF NOT heating_mode THEN  SPALNYA_HVAC.klapan:=16#7FFF; ELSE SPALNYA_HVAC.klapan:=16#0;END_IF
		END_CASE
	END_IF

	IF SPALNYA_HVAC.heat_mode=3 THEN (*fan*)
		SPALNYA_HVAC.tepla_pidloga:=FALSE;
		CASE SPALNYA_HVAC.heat_speed OF
			1:	SPALNYA_HVAC.fancoil_speed:=0;
				SPALNYA_HVAC.zaslinka:=TRUE;(*closed*)
				SPALNYA_HVAC.klapan:=16#0;(*full closed*)
			2:	SPALNYA_HVAC.fancoil_speed:=2;
				SPALNYA_HVAC.zaslinka:=FALSE;(*opened*)
				SPALNYA_HVAC.klapan:=16#0;
			3:	SPALNYA_HVAC.fancoil_speed:=3;
				SPALNYA_HVAC.zaslinka:=FALSE;(*opened*)
				SPALNYA_HVAC.klapan:=16#0;
		END_CASE
		IF heat.t_out<0 THEN SPALNYA_HVAC.klapan:=16#3FFF;(*30%*) ELSE SPALNYA_HVAC.klapan:=16#0;END_IF
	END_IF
END_PROGRAM

(* POU HVAC/winter, ST *)
PROGRAM winter
VAR

END_VAR
(*1-COOL mode 2-HEAT mode, 3-FAN mode*)

(*--------------------------VITALNYA---------------------------------------------------------------*)

	IF VITALNYA_HVAC.heat_mode=2 THEN
				VITALNYA_HVAC.zaslinka:=TRUE;(*closed*)
				VITALNYA_HVAC.tepla_pidloga:=TRUE; (*all opened*)
		CASE VITALNYA_HVAC.heat_speed OF

			1:	VITALNYA_HVAC.fancoil_speed:=1;
				VITALNYA_HVAC.klapan:=16#3FFF;
			2:	VITALNYA_HVAC.fancoil_speed:=2;
				VITALNYA_HVAC.klapan:=16#5FFF;
			3:	VITALNYA_HVAC.fancoil_speed:=3;
				VITALNYA_HVAC.klapan:=16#7FFF;
		END_CASE
	END_IF

	IF VITALNYA_HVAC.heat_mode=1 THEN
				VITALNYA_HVAC.klapan:=16#0;(*full closed*)
				VITALNYA_HVAC.zaslinka:=FALSE;
				VITALNYA_HVAC.tepla_pidloga:=FALSE; (*all closed*)

			CASE VITALNYA_HVAC.heat_speed OF
			1:	VITALNYA_HVAC.fancoil_speed:=1;
			2:	VITALNYA_HVAC.fancoil_speed:=2;
			3:	VITALNYA_HVAC.fancoil_speed:=3;
		END_CASE
	END_IF

	IF VITALNYA_HVAC.heat_mode=3 THEN
		VITALNYA_HVAC.tepla_pidloga:=FALSE;
		IF heat.t_out<0 THEN VITALNYA_HVAC.klapan:=16#3FFF;(*30%*) ELSE VITALNYA_HVAC.klapan:=16#0;END_IF
		CASE VITALNYA_HVAC.heat_speed OF
			1:	VITALNYA_HVAC.fancoil_speed:=0;
				VITALNYA_HVAC.zaslinka:=TRUE;(*closed*)
				VITALNYA_HVAC.klapan:=16#0;(*full closed*)
			2:	VITALNYA_HVAC.fancoil_speed:=2;
				VITALNYA_HVAC.zaslinka:=FALSE;(*opened*)
			3:	VITALNYA_HVAC.fancoil_speed:=3;
				VITALNYA_HVAC.zaslinka:=FALSE;(*opened*)
		END_CASE
	END_IF



(*--------------------------KABINET---------------------------------------------------------------*)
(*реверс двигуна клапана*)

	IF KABINET_HVAC.heat_mode=2 THEN
				KABINET_HVAC.zaslinka:=TRUE;(*closed*)
				KABINET_HVAC.tepla_pidloga:=TRUE; (*all opened*)
		CASE KABINET_HVAC.heat_speed OF

			1:	KABINET_HVAC.fancoil_speed:=1;
				KABINET_HVAC.klapan:=16#5FFF;
			2:	KABINET_HVAC.fancoil_speed:=2;
				KABINET_HVAC.klapan:=16#3FFF;
			3:	KABINET_HVAC.fancoil_speed:=3;
				KABINET_HVAC.klapan:=16#1FFF;
		END_CASE
	END_IF

	IF KABINET_HVAC.heat_mode=1 THEN
				KABINET_HVAC.klapan:=16#7FFF;(*full closed*)
				KABINET_HVAC.zaslinka:=FALSE;
				KABINET_HVAC.tepla_pidloga:=FALSE; (*all closed*)

			CASE KABINET_HVAC.heat_speed OF
			1:	KABINET_HVAC.fancoil_speed:=1;
			2:	KABINET_HVAC.fancoil_speed:=2;
			3:	KABINET_HVAC.fancoil_speed:=3;
		END_CASE
	END_IF

	IF KABINET_HVAC.heat_mode=3 THEN
		KABINET_HVAC.tepla_pidloga:=FALSE;
		IF heat.t_out<0 THEN KABINET_HVAC.klapan:=16#5FFF;(*30%*) ELSE KABINET_HVAC.klapan:=16#7FFF;END_IF
		CASE KABINET_HVAC.heat_speed OF
			1:	KABINET_HVAC.fancoil_speed:=0;
				KABINET_HVAC.zaslinka:=TRUE;(*closed*)
				KABINET_HVAC.klapan:=16#7FFF;(*full closed*)
			2:	KABINET_HVAC.fancoil_speed:=2;
				KABINET_HVAC.zaslinka:=FALSE;(*opened*)
			3:	KABINET_HVAC.fancoil_speed:=3;
				KABINET_HVAC.zaslinka:=FALSE;(*opened*)
		END_CASE
	END_IF



(*--------------------------KINO---------------------------------------------------------------*)
(*реверс двигуна клапана*)
	IF KINO_HVAC.heat_mode=2 THEN
				KINO_HVAC.zaslinka:=TRUE;(*closed*)
				KINO_HVAC.tepla_pidloga:=TRUE; (*all opened*)
		CASE KINO_HVAC.heat_speed OF

			1:	KINO_HVAC.fancoil_speed:=1;
				KINO_HVAC.klapan:=16#5FFF;
			2:	KINO_HVAC.fancoil_speed:=2;
				KINO_HVAC.klapan:=16#3FFF;
			3:	KINO_HVAC.fancoil_speed:=3;
				KINO_HVAC.klapan:=16#1FFF;
		END_CASE
	END_IF

	IF KINO_HVAC.heat_mode=1 THEN
				KINO_HVAC.klapan:=16#0;(*full closed*)
				KINO_HVAC.zaslinka:=FALSE;
				KINO_HVAC.tepla_pidloga:=FALSE; (*all closed*)

			CASE KINO_HVAC.heat_speed OF
			1:	KINO_HVAC.fancoil_speed:=1;
			2:	KINO_HVAC.fancoil_speed:=2;
			3:	KINO_HVAC.fancoil_speed:=3;
		END_CASE
	END_IF

	IF KINO_HVAC.heat_mode=3 THEN
		KINO_HVAC.tepla_pidloga:=FALSE;
		IF heat.t_out<0 THEN KINO_HVAC.klapan:=16#5FFF;(*30%*) ELSE KINO_HVAC.klapan:=16#7FFF;END_IF
		CASE KINO_HVAC.heat_speed OF
			1:	KINO_HVAC.fancoil_speed:=0;
				KINO_HVAC.zaslinka:=TRUE;(*closed*)
				KINO_HVAC.klapan:=16#7FFF;(*full closed*)
			2:	KINO_HVAC.fancoil_speed:=2;
				KINO_HVAC.zaslinka:=FALSE;(*opened*)
			3:	KINO_HVAC.fancoil_speed:=3;
				KINO_HVAC.zaslinka:=FALSE;(*opened*)
		END_CASE
	END_IF



(*--------------------------DYTJACHA---------------------------------------------------------------*)
(*реверс двигуна клапана*)
	IF DYTJACHA_HVAC.heat_mode=2 THEN
				DYTJACHA_HVAC.zaslinka:=TRUE;(*closed*)
				DYTJACHA_HVAC.tepla_pidloga:=TRUE; (*all opened*)
		CASE DYTJACHA_HVAC.heat_speed OF

			1:	DYTJACHA_HVAC.fancoil_speed:=1;
				DYTJACHA_HVAC.klapan:=16#5FFF;
			2:	DYTJACHA_HVAC.fancoil_speed:=2;
				DYTJACHA_HVAC.klapan:=16#3FFF;
			3:	DYTJACHA_HVAC.fancoil_speed:=3;
				DYTJACHA_HVAC.klapan:=16#1FFF;
		END_CASE
	END_IF

	IF DYTJACHA_HVAC.heat_mode=1 THEN
				DYTJACHA_HVAC.klapan:=16#7FFF;(*full closed*)
				DYTJACHA_HVAC.zaslinka:=FALSE;
				DYTJACHA_HVAC.tepla_pidloga:=FALSE; (*all closed*)

			CASE DYTJACHA_HVAC.heat_speed OF
			1:	DYTJACHA_HVAC.fancoil_speed:=1;
			2:	DYTJACHA_HVAC.fancoil_speed:=2;
			3:	DYTJACHA_HVAC.fancoil_speed:=3;
		END_CASE
	END_IF

	IF DYTJACHA_HVAC.heat_mode=3 THEN
		DYTJACHA_HVAC.tepla_pidloga:=FALSE;
		IF heat.t_out<0 THEN DYTJACHA_HVAC.klapan:=16#5FFF;(*30%*) ELSE DYTJACHA_HVAC.klapan:=16#7FFF;END_IF
		CASE DYTJACHA_HVAC.heat_speed OF
			1:	DYTJACHA_HVAC.fancoil_speed:=0;
				DYTJACHA_HVAC.zaslinka:=TRUE;(*closed*)
				DYTJACHA_HVAC.klapan:=16#7FFF;(*full closed*)
			2:	DYTJACHA_HVAC.fancoil_speed:=2;
				DYTJACHA_HVAC.zaslinka:=FALSE;(*opened*)
			3:	DYTJACHA_HVAC.fancoil_speed:=3;
				DYTJACHA_HVAC.zaslinka:=FALSE;(*opened*)
		END_CASE
	END_IF



(*--------------------------SPALNYA---------------------------------------------------------------*)

	IF SPALNYA_HVAC.heat_mode=2 THEN
				SPALNYA_HVAC.zaslinka:=TRUE;(*closed*)
				SPALNYA_HVAC.tepla_pidloga:=TRUE; (*all opened*)
		CASE SPALNYA_HVAC.heat_speed OF

			1:	SPALNYA_HVAC.fancoil_speed:=1;
				SPALNYA_HVAC.klapan:=16#3FFF;
			2:	SPALNYA_HVAC.fancoil_speed:=2;
				SPALNYA_HVAC.klapan:=16#5FFF;
			3:	SPALNYA_HVAC.fancoil_speed:=3;
				SPALNYA_HVAC.klapan:=16#7FFF;
		END_CASE
	END_IF

	IF SPALNYA_HVAC.heat_mode=1 THEN
				SPALNYA_HVAC.klapan:=16#0;(*full closed*)
				SPALNYA_HVAC.zaslinka:=FALSE;
				SPALNYA_HVAC.tepla_pidloga:=FALSE; (*all closed*)

			CASE SPALNYA_HVAC.heat_speed OF
			1:	SPALNYA_HVAC.fancoil_speed:=1;
			2:	SPALNYA_HVAC.fancoil_speed:=2;
			3:	SPALNYA_HVAC.fancoil_speed:=3;
		END_CASE
	END_IF

	IF SPALNYA_HVAC.heat_mode=3 THEN
		SPALNYA_HVAC.tepla_pidloga:=FALSE;
		IF heat.t_out<0 THEN SPALNYA_HVAC.klapan:=16#3FFF;(*30%*) ELSE SPALNYA_HVAC.klapan:=16#0;END_IF
		CASE SPALNYA_HVAC.heat_speed OF
			1:	SPALNYA_HVAC.fancoil_speed:=0;
				SPALNYA_HVAC.zaslinka:=TRUE;(*closed*)
				SPALNYA_HVAC.klapan:=16#0;(*full closed*)
			2:	SPALNYA_HVAC.fancoil_speed:=2;
				SPALNYA_HVAC.zaslinka:=FALSE;(*opened*)
			3:	SPALNYA_HVAC.fancoil_speed:=3;
				SPALNYA_HVAC.zaslinka:=FALSE;(*opened*)
		END_CASE
	END_IF
END_PROGRAM
